(* Schneider Machine Expert - Basic project Building, file version 2.9.0.0 *)
(* ProjectInformations: Name=BUILDING *)

HARDWARE
  Cpu 0: TM221CE40T
  EthernetConfiguration: NetworkName=M221, IpAllocationMode=FixedAddress, IpAddress=0.0.0.0, SubnetMask=0.0.0.0
  SerialLineConfiguration: Baud=Baud19200, Parity=ParityEven, DataBits=DataBits8, StopBits=StopBits1, PhysicalMedium=PhysicalMediumRs485, TransmissionMode=TransmissionModeModbusRtu, SlaveId=1, Addressing=SlaveAddressing
  MastTask: UsePeriodScanMode=false, PeriodScan=100
  FastTask: Period=255
  CpuBehavior: StartingMode=StartAsPreviousState, AutoSaveRamOnEeprom=true, WatchdogPeriod=250

SYMBOLS  (address, symbol, comment, settings)
  %M0       NWDAY_HEAT_ENABLE
  %M1       WORK_MON
  %M2       WORK_TUE
  %M3       WORK_WED
  %M4       WORK_THU
  %M5       WORK_FRI
  %M6       WORK_SAT
  %M7       WORK_SUN
  %M8       IS_WORK_DAY
  %M9       IS_COLD_MONTH
  %M10      RTC_SHIFTED_FW
  %M11      RTC_SHIFTED_BW
  %M12      BEGIN_RTC_TIME_SHIFT
  %M13      INSIDE_PCYCLE
  %M14      OUTSIDE_PCYCLE
  %M17      PLOT_FULL
  %M18      ARMING
  %M19      ARMED
  %M20      TRIGGERED
  %M25      FOPEN_MAIN_DOOR  "FORCES OPEN LOBBY DOOR"
  %M26      FS_TESTING_MODE  "DISABLES CALLING FIREMEN"
  %M27      SS_TESTING_MODE  "DISABLES CALLING SECURITY"
  %M28      AUTO_LIGHTS_L
  %M29      WDONLY_LIGHTS_L  "WORK DAYS ONLY"
  %M30      BTN_ENABLE_LIGHTS_L
  %M32      AUTO_MODE_LIGHTS_L  "1=MOVEMENT 0=KEEP_ON"
  %M33      CHANGED_LIGHTS_L
  %M34      MOVEMENT_LIGHTS_L
  %M35      AUTO_LIGHTS_B
  %M36      WDONLY_LIGHTS_B
  %M37      BTN_ENABLE_LIGHTS_B
  %M39      AUTO_MODE_LIGHTS_B
  %M40      CHANGED_LIGHTS_B
  %M41      MOVEMENT_LIGHTS_B
  %M100     RFID1_REQUEST
  %M101     RFID1_RESPONSE
  %M102     RFID1_ACCEPT
  %M103     RFID1_DENIED
  %M106     RFID2_REQUEST
  %M107     RFID2_RESPONSE
  %M108     RFID2_ACCEPT
  %M109     RFID2_DENIED
  %M112     RFID3_REQUEST
  %M113     RFID3_RESPONSE
  %M114     RFID3_ACCEPT
  %M115     RFID3_DENIED
  %M118     RFID4_REQUEST
  %M119     RFID4_RESPONSE
  %M120     RFID4_ACCEPT
  %M121     RFID4_DENIED
  %M124     RFID5_REQUEST
  %M125     RFID5_RESPONSE
  %M126     PGATE_ACCEPT  "RFID5_ACCEPT"
  %M127     RFID5_DENIED
  %M128     PGATE_FOPEN  "FORCE OPEN"
  %M129     PGATE_FCLOSE  "FORCE CLOSE"
  %M199     SIM_IO  "DISABLES REAL IO"
  %M200     I00  "O3_HEATER_ENABLE"
  %M201     I01  "O3_COOLER_ENABLE"
  %M202     I02  "L_DOOR_OPENED"
  %M203     I03  "O1_DOOR_OPENED"
  %M204     I04  "O2_DOOR_OPENED"
  %M205     I05  "O3_DOOR_OPENED"
  %M206     I06  "P_GATE_OPENED"
  %M207     I07  "P_GATE_CLOSED"
  %M208     I08  "P_GATE_OBJECT"
  %M209     I09  "P_GATE_BTN"
  %M210     I10  "L_MAN_LIGHT"
  %M211     I11  "B_MAN_LIGHT"
  %M212     I12  "L_MOTION"
  %M213     I13  "C_MOTION"
  %M214     I14  "O_MOTION"
  %M215     I15  "SECURITY_KEY"
  %M216     I16  "F_ALARM_BTN"
  %M217     I17  "F_ALARM_STOP"
  %M218     I18  "O1_SMOKE"
  %M219     I19  "O2_SMOKE"
  %M220     I20  "O3_SMOKE"
  %M221     I21  "L_SMOKE"
  %M222     I22  "C1_SMOKE"
  %M223     I23  "C2_SMOKE"
  %M224     Q00  "FIRE_SIREN"
  %M225     PWM1_IN  "SCRTY_BUZZER"
  %M226     Q02  "RFID1_UNLOCK"
  %M227     Q03  "RFID2_UNLOCK"
  %M228     Q04  "RFID3_UNLOCK"
  %M229     Q05  "RFID4_UNLOCK"
  %M230     Q06  "PGATE_OPEN"
  %M231     Q07  "PGATE_CLOSE"
  %M232     Q08  "HEATER"
  %M233     Q09  "COOLER"
  %M234     Q10  "LIGHTS_L"
  %M235     Q11  "LIGHTS_B"
  %M236     Q12  "SPRINKLERS"
  %M237     Q13  "DIAL_SECURITY"
  %M238     Q14  "DIAL_FIREMEN"
  %M239     Q15  "PGATE_BULB"
  %M495     WARNING_CONFIG_ALTERED
  %M496     WARNING_AUTOSEC_IMPOSSIBLE
  %M497     WARNING_FIRE_DETECTED
  %M498     WARNING_PGATE_OPENED  "OUTSIDE PARKING CYCLE"
  %M499     WARNING_PSPOT_MISCOUNT
  %M505     ERROR_LIGHT_CONFIG
  %M506     ERROR_PGATE_FCLOPEN
  %M507     ERROR_PARKING_SPOT_CONFIG
  %M508     ERROR_TEMP_CONFIG
  %M509     ERROR_WORK_DAY_CONFIG
  %M510     ERROR_COLD_MONTH_CONFIG
  %M511     EMERGENCY
  %S50      SB_RTCUPDATE  "Set to 1, this bit allows to update the date and time"
  %SW51     SW_RTCHHMM  "RTC Function: contains in BCD HHMM: hour and minute"
  %MW0      DESIRED_TEMP
  %MW1      TOLERANCE_TEMP
  %MW2      NWDAY_DESIRED_TEMP
  %MW3      WORK_DAY_START
  %MW4      WORK_DAY_END
  %MW5      COLD_MONTH_START
  %MW6      COLD_MONTH_END
  %MW7      RTC_DESIRED_HOUR
  %MW8      PARKING_SPOT_COUNT
  %MW9      PARKING_SPOTS_TAKEN
  %MW10     PARKING_SPOT_THCOUNT  "THEORETICAL COUNT ~= <P_LOT_AREA>/11,5 (m^2)"
  %MW11     PGATE_PASSED_OBJECTS
  %MW12     PGATE_UNAUTH_OBJECTS
  %MW13     ACTIVE_SMOKE_COUNT
  %MW14     TRESHOLD_LIGHTS
  %MW15     TOLERANCE_LIGHTS
  %MW100    RFID1_REQ_START
  %MW101    RFID1_REQ_MID
  %MW102    RFID1_REQ_END
  %MW103    RFID1_RESP_START
  %MW104    RFID1_RESP_MID
  %MW105    RFID1_RESP_END
  %MW106    RFID2_REQ_START
  %MW107    RFID2_REQ_MID
  %MW108    RFID2_REQ_END
  %MW109    RFID2_RESP_START
  %MW110    RFID2_RESP_MID
  %MW111    RFID2_RESP_END
  %MW112    RFID3_REQ_START
  %MW113    RFID3_REQ_MID
  %MW114    RFID3_REQ_END
  %MW115    RFID3_RESP_START
  %MW116    RFID3_RESP_MID
  %MW117    RFID3_RESP_END
  %MW118    RFID4_REQ_START
  %MW119    RFID4_REQ_MID
  %MW120    RFID4_REQ_END
  %MW121    RFID4_RESP_START
  %MW122    RFID4_RESP_MID
  %MW123    RFID4_RESP_END
  %MW124    RFID5_REQ_START
  %MW125    RFID5_REQ_MID
  %MW126    RFID5_REQ_END
  %MW127    RFID5_RESP_START
  %MW128    RFID5_RESP_MID
  %MW129    RFID5_RESP_END
  %MW200    IW0  "MEASURED_TEMP"
  %MW201    IW1  "MEASURED_LIGHT"
  %TM0      RFID1_TM  [Type=TP, Preset=30, Base=OneHundredMilliSeconds]
  %TM1      RFID2_TM  [Type=TP, Preset=30, Base=OneHundredMilliSeconds]
  %TM2      RFID3_TM  [Type=TP, Preset=30, Base=OneHundredMilliSeconds]
  %TM3      RFID4_TM  [Type=TP, Preset=30, Base=OneHundredMilliSeconds]
  %TM4      PGATE_TM  [Preset=200, Base=OneHundredMilliSeconds]
  %TM5      ARM_TM  "60s"  [Preset=600, Base=OneHundredMilliSeconds]
  %TM6      TRIG_TM  "45s"  [Preset=450, Base=OneHundredMilliSeconds]
  %TM8      LIGHT_TM_L  [Type=TP, Preset=600, Base=OneHundredMilliSeconds]
  %TM9      LIGHT_TM_B  [Type=TP, Preset=600, Base=OneHundredMilliSeconds]
  %RTC0     RTC  [Day(Value(int=25)), Month(Value(int=3)), Year(Value(int=2000)), Hours(Value(int=0)), Minutes(Value(int=0)), Seconds(Value(int=0))]
  %I0.0     O3_HEATER_ENABLE  "OFFICE3 FL2"
  %I0.1     O3_COOLER_ENABLE  "OFFICE3 FL2"
  %I0.2     L_DOOR_OPENED  "LOBBY FL0"
  %I0.3     O1_DOOR_OPENED  "OFFICE1 FL1"
  %I0.4     O2_DOOR_OPENED  "OFFICE2 FL1"
  %I0.5     O3_DOOR_OPENED  "OFFICE3 FL3"
  %I0.6     P_GATE_OPENED  "FULLY OPENED"
  %I0.7     P_GATE_CLOSED  "FULLY CLOSED"
  %I0.8     P_GATE_OBJECT  "DETECTED OBJECT"
  %I0.9     P_GATE_BTN  "INSIDE PARKING LOT"
  %I0.10    L_MAN_LIGHT  "LOBBY"
  %I0.11    B_MAN_LIGHT  "B = C1 + C2"
  %I0.12    L_MOTION  "LOBBY SECURITY LIGHTS"
  %I0.13    C_MOTION  "CORRIDORS SECURITY LIGHTS"
  %I0.14    O_MOTION  "OFFICES SECURITY ONLY"
  %I0.15    SECURITY_KEY  "LOBBY FL0"
  %I0.16    F_ALARM_BTN  "FL0 FL1 FL2"
  %I0.17    F_ALARM_STOP  "FL0 FL1 FL2"
  %I0.18    O1_SMOKE  "OFFICE1 F1"
  %I0.19    O2_SMOKE  "OFFICE2 FL1"
  %I0.20    O3_SMOKE  "OFFICE3 FL2"
  %I0.21    L_SMOKE  "LOBBY FL0"
  %I0.22    C1_SMOKE  "CORRIDOR1 FL1"
  %I0.23    C2_SMOKE  "CORRIDOR2 FL2"
  %Q0.0     FIRE_SIREN
  %Q0.1     SCRTY_BUZZER
  %Q0.2     RFID1_UNLOCK  "LOBBY FL0"
  %Q0.3     RFID2_UNLOCK  "O1 FL1"
  %Q0.4     RFID3_UNLOCK  "O2 FL2"
  %Q0.5     RFID4_UNLOCK  "O3 FL3"
  %Q0.6     PGATE_OPEN  "PARKING LOT"
  %Q0.7     PGATE_CLOSE  "PARKING LOT"
  %Q0.8     HEATER  "O3 FL2"
  %Q0.9     COOLER  "O3 FL2"
  %Q0.10    LIGHTS_L  "LOBBY FL0"
  %Q0.11    LIGHTS_B  "B = C1 + C2"
  %Q0.12    SPRINKLERS
  %Q0.13    DIAL_SECURITY
  %Q0.14    DIAL_FIREMEN
  %Q0.15    PGATE_BULB  "IN FRONT OF PARKING LOT GATE"
  %IW0.0    MEASURED_TEMP  "-50C to +50C"  [Type=Type_0_10V, Scope=Scope_Normal, Minimum=0, Maximum=1000]
  %IW0.1    MEASURED_LIGHT  [Type=Type_0_10V, Scope=Scope_Normal, Minimum=0, Maximum=1000]
  %PWM1     BUZZER  "2kHz"  [PtoObject(RefInput=NotUsed, ZPhaseInput=NotUsed, ProbeInput=NotUsed), GlobalIndex=1, Type=PWM, TimeBase=ZeroPointOneMilliSeconds, Preset=5]

POU MAIN
  (* SectionNumber=1 *)

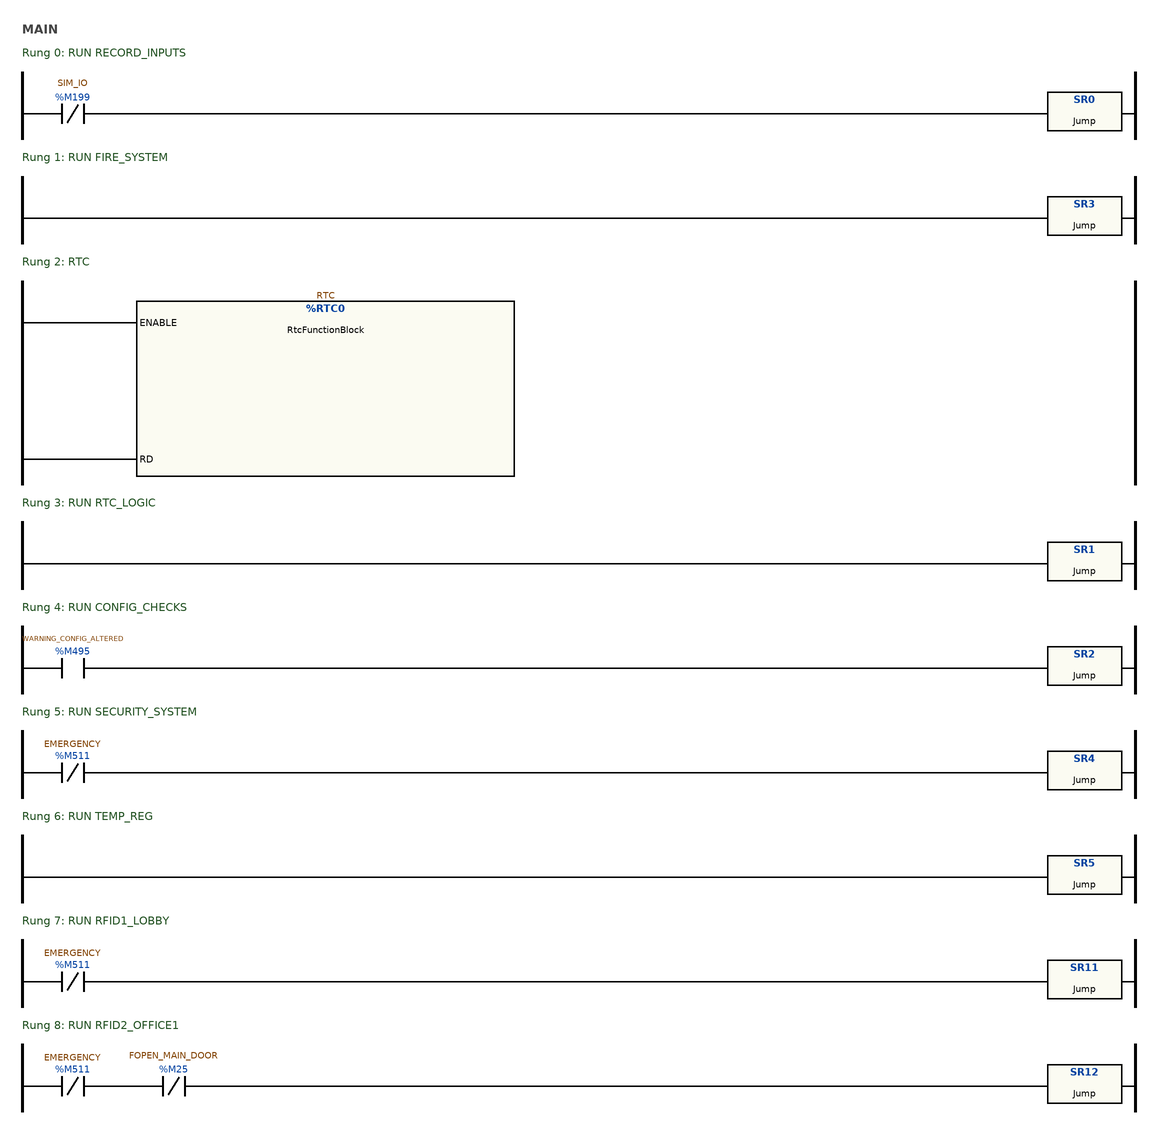

// Rung 0: RUN RECORD_INPUTS
  LDN %M199               (* SIM_IO *)
  SR0
  // as ST:
  //   IF NOT SIM_IO THEN SR0(); END_IF;

// Rung 1: RUN FIRE_SYSTEM
  LD 1
  SR3
  // as ST:
  //   SR3();

// Rung 2: RTC
  BLK %RTC0               (* RTC *)
  LD 1
  ENABLE
  LD 1
  RD
  END_BLK
  // as ST:
  //   RTC(ENABLE := TRUE, RD := TRUE);

// Rung 3: RUN RTC_LOGIC
  LD 1
  SR1
  // as ST:
  //   SR1();

// Rung 4: RUN CONFIG_CHECKS
  LD %M495                (* WARNING_CONFIG_ALTERED *)
  SR2
  // as ST:
  //   IF WARNING_CONFIG_ALTERED THEN SR2(); END_IF;

// Rung 5: RUN SECURITY_SYSTEM
  LDN %M511               (* EMERGENCY *)
  SR4
  // as ST:
  //   IF NOT EMERGENCY THEN SR4(); END_IF;

// Rung 6: RUN TEMP_REG
  LD 1
  SR5
  // as ST:
  //   SR5();

// Rung 7: RUN RFID1_LOBBY
  LDN %M511               (* EMERGENCY *)
  SR11
  // as ST:
  //   IF NOT EMERGENCY THEN SR11(); END_IF;

// Rung 8: RUN RFID2_OFFICE1
  LDN %M511               (* EMERGENCY *)
  ANDN %M25               (* FOPEN_MAIN_DOOR *)
  SR12
  // as ST:
  //   IF NOT EMERGENCY AND NOT FOPEN_MAIN_DOOR THEN SR12(); END_IF;

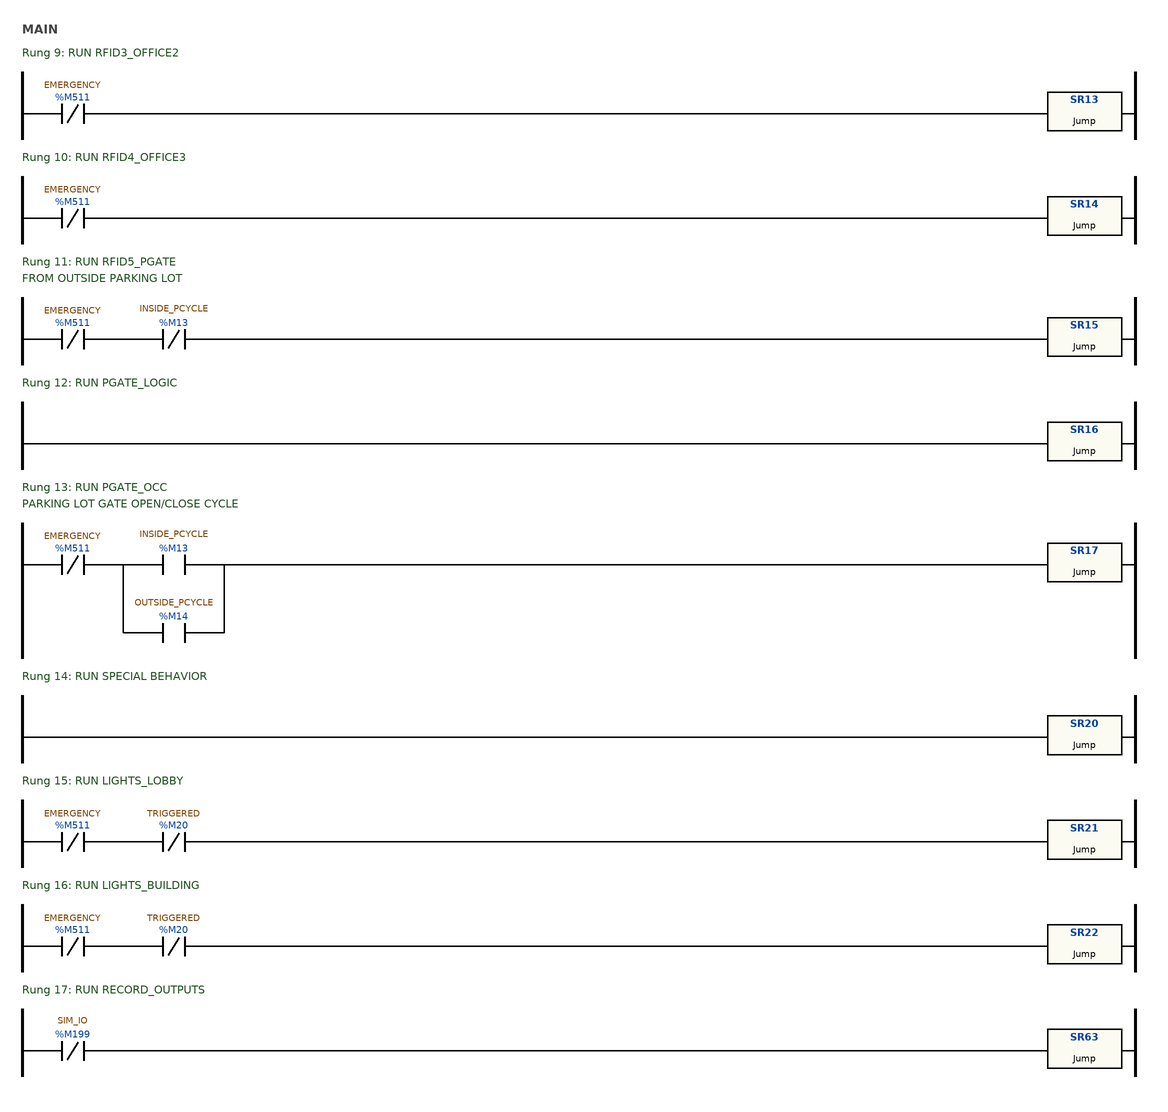

// Rung 9: RUN RFID3_OFFICE2
  LDN %M511               (* EMERGENCY *)
  SR13
  // as ST:
  //   IF NOT EMERGENCY THEN SR13(); END_IF;

// Rung 10: RUN RFID4_OFFICE3
  LDN %M511               (* EMERGENCY *)
  SR14
  // as ST:
  //   IF NOT EMERGENCY THEN SR14(); END_IF;

// Rung 11: RUN RFID5_PGATE
// FROM OUTSIDE PARKING LOT
  LDN %M511               (* EMERGENCY *)
  ANDN %M13               (* INSIDE_PCYCLE *)
  SR15
  // as ST:
  //   IF NOT EMERGENCY AND NOT INSIDE_PCYCLE THEN SR15(); END_IF;

// Rung 12: RUN PGATE_LOGIC
  LD 1
  SR16
  // as ST:
  //   SR16();

// Rung 13: RUN PGATE_OCC
// PARKING LOT GATE OPEN/CLOSE CYCLE
  LDN %M511               (* EMERGENCY *)
  AND( %M13               (* INSIDE_PCYCLE *)
  OR %M14                 (* OUTSIDE_PCYCLE *)
  )
  SR17
  // as ST:
  //   IF NOT EMERGENCY AND (INSIDE_PCYCLE OR OUTSIDE_PCYCLE) THEN SR17(); END_IF;

// Rung 14: RUN SPECIAL BEHAVIOR
  LD 1
  SR20
  // as ST:
  //   SR20();

// Rung 15: RUN LIGHTS_LOBBY
  LDN %M511               (* EMERGENCY *)
  ANDN %M20               (* TRIGGERED *)
  SR21
  // as ST:
  //   IF NOT EMERGENCY AND NOT TRIGGERED THEN SR21(); END_IF;

// Rung 16: RUN LIGHTS_BUILDING
  LDN %M511               (* EMERGENCY *)
  ANDN %M20               (* TRIGGERED *)
  SR22
  // as ST:
  //   IF NOT EMERGENCY AND NOT TRIGGERED THEN SR22(); END_IF;

// Rung 17: RUN RECORD_OUTPUTS
  LDN %M199               (* SIM_IO *)
  SR63
  // as ST:
  //   IF NOT SIM_IO THEN SR63(); END_IF;

Subroutine RECORD_INPUTS
  (* SectionNumber=2, Number=0 *)

// Rung 18: %I0.0 TO I00
  LD %I0.0                (* O3_HEATER_ENABLE *)
  ST %M200                (* I00 *)
  // as ST:
  //   I00 := O3_HEATER_ENABLE;

// Rung 19: %I0.1 TO I01
  LD %I0.1                (* O3_COOLER_ENABLE *)
  ST %M201                (* I01 *)
  // as ST:
  //   I01 := O3_COOLER_ENABLE;

// Rung 20: %I0.2 TO I02
  LD %I0.2                (* L_DOOR_OPENED *)
  ST %M202                (* I02 *)
  // as ST:
  //   I02 := L_DOOR_OPENED;

// Rung 21: %I0.3 TO I03
  LD %I0.3                (* O1_DOOR_OPENED *)
  ST %M203                (* I03 *)
  // as ST:
  //   I03 := O1_DOOR_OPENED;

// Rung 22: %I0.4 TO I04
  LD %I0.4                (* O2_DOOR_OPENED *)
  ST %M204                (* I04 *)
  // as ST:
  //   I04 := O2_DOOR_OPENED;

// Rung 23: %I0.5 TO I05
  LD %I0.5                (* O3_DOOR_OPENED *)
  ST %M205                (* I05 *)
  // as ST:
  //   I05 := O3_DOOR_OPENED;

// Rung 24: %I0.6 TO I06
  LD %I0.6                (* P_GATE_OPENED *)
  ST %M206                (* I06 *)
  // as ST:
  //   I06 := P_GATE_OPENED;

// Rung 25: %I0.7 TO I07
  LD %I0.7                (* P_GATE_CLOSED *)
  ST %M207                (* I07 *)
  // as ST:
  //   I07 := P_GATE_CLOSED;

// Rung 26: %I0.8 TO I08
  LD %I0.8                (* P_GATE_OBJECT *)
  ST %M208                (* I08 *)
  // as ST:
  //   I08 := P_GATE_OBJECT;

// Rung 27: %I0.9 TO I09
  LD %I0.9                (* P_GATE_BTN *)
  ST %M209                (* I09 *)
  // as ST:
  //   I09 := P_GATE_BTN;

// Rung 28: %I0.10 TO I10
  LD %I0.10               (* L_MAN_LIGHT *)
  ST %M210                (* I10 *)
  // as ST:
  //   I10 := L_MAN_LIGHT;

// Rung 29: %I0.11 TO I11
  LD %I0.11               (* B_MAN_LIGHT *)
  ST %M211                (* I11 *)
  // as ST:
  //   I11 := B_MAN_LIGHT;

// Rung 30: %I0.12 TO I12
  LD %I0.12               (* L_MOTION *)
  ST %M212                (* I12 *)
  // as ST:
  //   I12 := L_MOTION;

// Rung 31: %I0.13 TO I13
  LD %I0.13               (* C_MOTION *)
  ST %M213                (* I13 *)
  // as ST:
  //   I13 := C_MOTION;

// Rung 32: %I0.14 TO I14
  LD %I0.14               (* O_MOTION *)
  ST %M214                (* I14 *)
  // as ST:
  //   I14 := O_MOTION;

// Rung 33: %I0.15 TO I15
  LD %I0.15               (* SECURITY_KEY *)
  ST %M215                (* I15 *)
  // as ST:
  //   I15 := SECURITY_KEY;

// Rung 34: %I0.16 TO I16
  LD %I0.16               (* F_ALARM_BTN *)
  ST %M216                (* I16 *)
  // as ST:
  //   I16 := F_ALARM_BTN;

// Rung 35: %I0.17 TO I17
  LD %I0.17               (* F_ALARM_STOP *)
  ST %M217                (* I17 *)
  // as ST:
  //   I17 := F_ALARM_STOP;

// Rung 36: %I0.18 TO I18
  LD %I0.18               (* O1_SMOKE *)
  ST %M218                (* I18 *)
  // as ST:
  //   I18 := O1_SMOKE;

// Rung 37: %I0.19 TO I19
  LD %I0.19               (* O2_SMOKE *)
  ST %M219                (* I19 *)
  // as ST:
  //   I19 := O2_SMOKE;

// Rung 38: %I0.20 TO I20
  LD %I0.20               (* O3_SMOKE *)
  ST %M220                (* I20 *)
  // as ST:
  //   I20 := O3_SMOKE;

// Rung 39: %I0.21 TO I21
  LD %I0.21               (* L_SMOKE *)
  ST %M221                (* I21 *)
  // as ST:
  //   I21 := L_SMOKE;

// Rung 40: %I0.22 TO I22
  LD %I0.22               (* C1_SMOKE *)
  ST %M222                (* I22 *)
  // as ST:
  //   I22 := C1_SMOKE;

// Rung 41: %I0.23 TO I23
  LD %I0.23               (* C2_SMOKE *)
  ST %M223                (* I23 *)
  // as ST:
  //   I23 := C2_SMOKE;

// Rung 42: %IW0.0 TO IW0
  LD 1
  [ %MW200 := %IW0.0 ]    (* IW0, MEASURED_TEMP *)
  // as ST:
  //   IW0 := MEASURED_TEMP;

// Rung 43: %IW0.1 TO IW1
  LD 1
  [ %MW201 := %IW0.1 ]    (* IW1, MEASURED_LIGHT *)
  // as ST:
  //   IW1 := MEASURED_LIGHT;

Subroutine RTC_LOGIC
  (* SectionNumber=3, Number=1 *)

// Rung 44: RTC DST FORWARD SHIFT REQUEST
  LDN %M10                (* RTC_SHIFTED_FW *)
  AND [ %RTC0.HOURS = 3 ] (* RTC *)
  AND [ %RTC0.MINUTES = 0 ](* RTC *)
  AND [ %RTC0.SECONDS = 0 ](* RTC *)
  AND [ %RTC0.MONTH = 3 ] (* RTC *)
  AND [ %RTC0.DAY >= 25 ] (* RTC *)
  AND [ %RTC0.DAYOFWEEK = 7 ](* RTC *)
  S %M10                  (* RTC_SHIFTED_FW *)
  R %M11                  (* RTC_SHIFTED_BW *)
  [ %MW7 := 1024 ]        (* RTC_DESIRED_HOUR *)
  // as ST:
  //   _t1 := NOT RTC_SHIFTED_FW AND RTC.HOURS = 3 AND RTC.MINUTES = 0 AND RTC.SECONDS = 0 AND RTC.MONTH = 3 AND RTC.DAY >= 25 AND RTC.DAYOFWEEK = 7;
  //   IF _t1 THEN RTC_SHIFTED_FW := TRUE; END_IF;
  //   IF _t1 THEN RTC_SHIFTED_BW := FALSE; END_IF;
  //   IF _t1 THEN RTC_DESIRED_HOUR := 1024; END_IF;

// Rung 45: RTC DST BACKWARD SHIFT REQUEST
  LDN %M11                (* RTC_SHIFTED_BW *)
  AND [ %RTC0.HOURS = 4 ] (* RTC *)
  AND [ %RTC0.MINUTES = 0 ](* RTC *)
  AND [ %RTC0.SECONDS = 0 ](* RTC *)
  AND [ %RTC0.MONTH = 10 ](* RTC *)
  AND [ %RTC0.DAY >= 25 ] (* RTC *)
  AND [ %RTC0.DAYOFWEEK = 7 ](* RTC *)
  S %M11                  (* RTC_SHIFTED_BW *)
  R %M10                  (* RTC_SHIFTED_FW *)
  [ %MW7 := 768 ]         (* RTC_DESIRED_HOUR *)
  // as ST:
  //   _t1 := NOT RTC_SHIFTED_BW AND RTC.HOURS = 4 AND RTC.MINUTES = 0 AND RTC.SECONDS = 0 AND RTC.MONTH = 10 AND RTC.DAY >= 25 AND RTC.DAYOFWEEK = 7;
  //   IF _t1 THEN RTC_SHIFTED_BW := TRUE; END_IF;
  //   IF _t1 THEN RTC_SHIFTED_FW := FALSE; END_IF;
  //   IF _t1 THEN RTC_DESIRED_HOUR := 768; END_IF;

// Rung 46: RTC TIME SHIFT EXECUTE
  LDR %M10                (* RTC_SHIFTED_FW *)
  ORR %M11                (* RTC_SHIFTED_BW *)
  ST %S50                 (* SB_RTCUPDATE *)
  [ %SW51 := %MW7 ]       (* SW_RTCHHMM, RTC_DESIRED_HOUR *)
  // as ST:
  //   SB_RTCUPDATE := RISING(RTC_SHIFTED_FW) OR RISING(RTC_SHIFTED_BW);
  //   IF RISING(RTC_SHIFTED_FW) OR RISING(RTC_SHIFTED_BW) THEN SW_RTCHHMM := RTC_DESIRED_HOUR; END_IF;

// Rung 47: WORK DAY CHECK
  LDN %M509               (* ERROR_WORK_DAY_CONFIG *)
  AND( %M1                (* WORK_MON *)
  AND [ %RTC0.DAYOFWEEK = 1 ](* RTC *)
  OR( %M2                 (* WORK_TUE *)
  AND [ %RTC0.DAYOFWEEK = 2 ](* RTC *)
  )
  OR( %M3                 (* WORK_WED *)
  AND [ %RTC0.DAYOFWEEK = 3 ](* RTC *)
  )
  OR( %M4                 (* WORK_THU *)
  AND [ %RTC0.DAYOFWEEK = 4 ](* RTC *)
  )
  OR( %M5                 (* WORK_FRI *)
  AND [ %RTC0.DAYOFWEEK = 5 ](* RTC *)
  )
  OR( %M6                 (* WORK_SAT *)
  AND [ %RTC0.DAYOFWEEK = 6 ](* RTC *)
  )
  OR( %M7                 (* WORK_SUN *)
  AND [ %RTC0.DAYOFWEEK = 7 ](* RTC *)
  )
  )
  AND [ %RTC0.HOURS >= %MW3 ](* RTC, WORK_DAY_START *)
  AND [ %RTC0.HOURS <= %MW4 ](* RTC, WORK_DAY_END *)
  ST %M8                  (* IS_WORK_DAY *)
  // as ST:
  //   IS_WORK_DAY := NOT ERROR_WORK_DAY_CONFIG AND (WORK_MON AND RTC.DAYOFWEEK = 1 OR WORK_TUE AND RTC.DAYOFWEEK = 2 OR WORK_WED AND RTC.DAYOFWEEK = 3 OR WORK_THU AND RTC.DAYOFWEEK = 4 OR WORK_FRI AND RTC.DAYOFWEEK = 5 OR WORK_SAT AND RTC.DAYOFWEEK = 6 OR WORK_SUN AND RTC.DAYOFWEEK = 7) AND RTC.HOURS >= WORK_DAY_START AND RTC.HOURS <= WORK_DAY_END;

Subroutine CONFIG_CHECKS
  (* SectionNumber=4, Number=2 *)

// Rung 48: COLD MONTH CONFIG ERROR
  LD %M0                  (* NWDAY_HEAT_ENABLE *)
  MPS
  AND [ %MW5 >= 1 ]       (* COLD_MONTH_START *)
  AND [ %MW5 <= 12 ]      (* COLD_MONTH_START *)
  AND [ %MW6 >= 1 ]       (* COLD_MONTH_END *)
  AND [ %MW6 <= 12 ]      (* COLD_MONTH_END *)
  R %M510                 (* ERROR_COLD_MONTH_CONFIG *)
  MPP
  AND( [ %MW5 < 1 ]       (* COLD_MONTH_START *)
  OR [ %MW5 > 12 ]        (* COLD_MONTH_START *)
  OR [ %MW6 < 1 ]         (* COLD_MONTH_END *)
  OR [ %MW6 > 12 ]        (* COLD_MONTH_END *)
  )
  S %M510                 (* ERROR_COLD_MONTH_CONFIG *)
  // as ST:
  //   IF NWDAY_HEAT_ENABLE AND COLD_MONTH_START >= 1 AND COLD_MONTH_START <= 12 AND COLD_MONTH_END >= 1 AND COLD_MONTH_END <= 12 THEN ERROR_COLD_MONTH_CONFIG := FALSE; END_IF;
  //   IF NWDAY_HEAT_ENABLE AND (COLD_MONTH_START < 1 OR COLD_MONTH_START > 12 OR COLD_MONTH_END < 1 OR COLD_MONTH_END > 12) THEN ERROR_COLD_MONTH_CONFIG := TRUE; END_IF;

// Rung 49: WORK DAY CONFIG ERROR
  LD %M1                  (* WORK_MON *)
  OR %M2                  (* WORK_TUE *)
  OR %M3                  (* WORK_WED *)
  OR %M4                  (* WORK_THU *)
  OR %M5                  (* WORK_FRI *)
  OR %M6                  (* WORK_SAT *)
  OR %M7                  (* WORK_SUN *)
  MPS
  AND [ %MW3 > 0 ]        (* WORK_DAY_START *)
  AND [ %MW4 > 0 ]        (* WORK_DAY_END *)
  AND [ %MW3 < 24 ]       (* WORK_DAY_START *)
  AND [ %MW4 < 24 ]       (* WORK_DAY_END *)
  AND [ %MW3 <= %MW4 ]    (* WORK_DAY_START, WORK_DAY_END *)
  R %M509                 (* ERROR_WORK_DAY_CONFIG *)
  MPP
  AND( [ %MW3 < 0 ]       (* WORK_DAY_START *)
  OR [ %MW4 < 0 ]         (* WORK_DAY_END *)
  OR [ %MW3 >= 24 ]       (* WORK_DAY_START *)
  OR [ %MW4 >= 24 ]       (* WORK_DAY_END *)
  OR [ %MW3 > %MW4 ]      (* WORK_DAY_START, WORK_DAY_END *)
  )
  S %M509                 (* ERROR_WORK_DAY_CONFIG *)
  // as ST:
  //   IF (WORK_MON OR WORK_TUE OR WORK_WED OR WORK_THU OR WORK_FRI OR WORK_SAT OR WORK_SUN) AND WORK_DAY_START > 0 AND WORK_DAY_END > 0 AND WORK_DAY_START < 24 AND WORK_DAY_END < 24 AND WORK_DAY_START <= WORK_DAY_END THEN ERROR_WORK_DAY_CONFIG := FALSE; END_IF;
  //   IF (WORK_MON OR WORK_TUE OR WORK_WED OR WORK_THU OR WORK_FRI OR WORK_SAT OR WORK_SUN) AND (WORK_DAY_START < 0 OR WORK_DAY_END < 0 OR WORK_DAY_START >= 24 OR WORK_DAY_END >= 24 OR WORK_DAY_START > WORK_DAY_END) THEN ERROR_WORK_DAY_CONFIG := TRUE; END_IF;

// Rung 50: WORK DAY NOT CONFIGURED
  LDN %M1                 (* WORK_MON *)
  ANDN %M2                (* WORK_TUE *)
  ANDN %M3                (* WORK_WED *)
  ANDN %M4                (* WORK_THU *)
  ANDN %M5                (* WORK_FRI *)
  ANDN %M6                (* WORK_SAT *)
  ANDN %M7                (* WORK_SUN *)
  R %M509                 (* ERROR_WORK_DAY_CONFIG *)
  // as ST:
  //   IF NOT WORK_MON AND NOT WORK_TUE AND NOT WORK_WED AND NOT WORK_THU AND NOT WORK_FRI AND NOT WORK_SAT AND NOT WORK_SUN THEN ERROR_WORK_DAY_CONFIG := FALSE; END_IF;

// Rung 51: WORK DAY TEMP CONFIG ERROR
  LD %M1                  (* WORK_MON *)
  OR %M2                  (* WORK_TUE *)
  OR %M3                  (* WORK_WED *)
  OR %M4                  (* WORK_THU *)
  OR %M5                  (* WORK_FRI *)
  OR %M6                  (* WORK_SAT *)
  OR %M7                  (* WORK_SUN *)
  MPS
  AND [ %MW0 >= 0 ]       (* DESIRED_TEMP *)
  AND [ %MW0 <= 1000 ]    (* DESIRED_TEMP *)
  AND [ %MW0 + %MW1 <= 1000 ](* DESIRED_TEMP, TOLERANCE_TEMP *)
  AND [ %MW0 - %MW1 >= 0 ](* DESIRED_TEMP, TOLERANCE_TEMP *)
  R %M508                 (* ERROR_TEMP_CONFIG *)
  MPP
  AND( [ %MW0 < 0 ]       (* DESIRED_TEMP *)
  OR [ %MW0 > 1000 ]      (* DESIRED_TEMP *)
  OR [ %MW0 + %MW1 > 1000 ](* DESIRED_TEMP, TOLERANCE_TEMP *)
  OR [ %MW0 - %MW1 < 0 ]  (* DESIRED_TEMP, TOLERANCE_TEMP *)
  )
  S %M508                 (* ERROR_TEMP_CONFIG *)
  // as ST:
  //   IF (WORK_MON OR WORK_TUE OR WORK_WED OR WORK_THU OR WORK_FRI OR WORK_SAT OR WORK_SUN) AND DESIRED_TEMP >= 0 AND DESIRED_TEMP <= 1000 AND DESIRED_TEMP + TOLERANCE_TEMP <= 1000 AND DESIRED_TEMP - TOLERANCE_TEMP >= 0 THEN ERROR_TEMP_CONFIG := FALSE; END_IF;
  //   IF (WORK_MON OR WORK_TUE OR WORK_WED OR WORK_THU OR WORK_FRI OR WORK_SAT OR WORK_SUN) AND (DESIRED_TEMP < 0 OR DESIRED_TEMP > 1000 OR DESIRED_TEMP + TOLERANCE_TEMP > 1000 OR DESIRED_TEMP - TOLERANCE_TEMP < 0) THEN ERROR_TEMP_CONFIG := TRUE; END_IF;

// Rung 52: NON WORK DAY TEMP CONFIG ERROR
  LD %M0                  (* NWDAY_HEAT_ENABLE *)
  MPS
  AND [ %MW2 >= 0 ]       (* NWDAY_DESIRED_TEMP *)
  AND [ %MW2 <= 1000 ]    (* NWDAY_DESIRED_TEMP *)
  AND [ %MW2 + %MW1 <= 1000 ](* NWDAY_DESIRED_TEMP, TOLERANCE_TEMP *)
  AND [ %MW2 - %MW1 >= 0 ](* NWDAY_DESIRED_TEMP, TOLERANCE_TEMP *)
  R %M508                 (* ERROR_TEMP_CONFIG *)
  MPP
  AND( [ %MW2 < 0 ]       (* NWDAY_DESIRED_TEMP *)
  OR [ %MW2 > 1000 ]      (* NWDAY_DESIRED_TEMP *)
  OR [ %MW2 + %MW1 > 1000 ](* NWDAY_DESIRED_TEMP, TOLERANCE_TEMP *)
  OR [ %MW2 - %MW1 < 0 ]  (* NWDAY_DESIRED_TEMP, TOLERANCE_TEMP *)
  )
  S %M508                 (* ERROR_TEMP_CONFIG *)
  // as ST:
  //   IF NWDAY_HEAT_ENABLE AND NWDAY_DESIRED_TEMP >= 0 AND NWDAY_DESIRED_TEMP <= 1000 AND NWDAY_DESIRED_TEMP + TOLERANCE_TEMP <= 1000 AND NWDAY_DESIRED_TEMP - TOLERANCE_TEMP >= 0 THEN ERROR_TEMP_CONFIG := FALSE; END_IF;
  //   IF NWDAY_HEAT_ENABLE AND (NWDAY_DESIRED_TEMP < 0 OR NWDAY_DESIRED_TEMP > 1000 OR NWDAY_DESIRED_TEMP + TOLERANCE_TEMP > 1000 OR NWDAY_DESIRED_TEMP - TOLERANCE_TEMP < 0) THEN ERROR_TEMP_CONFIG := TRUE; END_IF;

// Rung 53: DESIRED LIGHT CONFIG ERROR
  LD %M28                 (* AUTO_LIGHTS_L *)
  OR %M35                 (* AUTO_LIGHTS_B *)
  MPS
  AND [ %MW14 >= 0 ]      (* TRESHOLD_LIGHTS *)
  AND [ %MW14 <= 1000 ]   (* TRESHOLD_LIGHTS *)
  AND [ %MW14 - %MW15 >= 0 ](* TRESHOLD_LIGHTS, TOLERANCE_LIGHTS *)
  AND [ %MW14 + %MW15 <= 1000 ](* TRESHOLD_LIGHTS, TOLERANCE_LIGHTS *)
  R %M505                 (* ERROR_LIGHT_CONFIG *)
  MPP
  AND( [ %MW14 < 0 ]      (* TRESHOLD_LIGHTS *)
  OR [ %MW14 > 1000 ]     (* TRESHOLD_LIGHTS *)
  OR [ %MW14 - %MW15 < 0 ](* TRESHOLD_LIGHTS, TOLERANCE_LIGHTS *)
  OR [ %MW14 + %MW15 > 1000 ](* TRESHOLD_LIGHTS, TOLERANCE_LIGHTS *)
  )
  S %M505                 (* ERROR_LIGHT_CONFIG *)
  // as ST:
  //   IF (AUTO_LIGHTS_L OR AUTO_LIGHTS_B) AND TRESHOLD_LIGHTS >= 0 AND TRESHOLD_LIGHTS <= 1000 AND TRESHOLD_LIGHTS - TOLERANCE_LIGHTS >= 0 AND TRESHOLD_LIGHTS + TOLERANCE_LIGHTS <= 1000 THEN ERROR_LIGHT_CONFIG := FALSE; END_IF;
  //   IF (AUTO_LIGHTS_L OR AUTO_LIGHTS_B) AND (TRESHOLD_LIGHTS < 0 OR TRESHOLD_LIGHTS > 1000 OR TRESHOLD_LIGHTS - TOLERANCE_LIGHTS < 0 OR TRESHOLD_LIGHTS + TOLERANCE_LIGHTS > 1000) THEN ERROR_LIGHT_CONFIG := TRUE; END_IF;

// Rung 54: PARKING SPOT CONFIG ERROR
  LD [ %MW8 > %MW10 ]     (* PARKING_SPOT_COUNT, PARKING_SPOT_THCOUNT *)
  OR [ %MW8 < 0 ]         (* PARKING_SPOT_COUNT *)
  OR [ %MW10 < 0 ]        (* PARKING_SPOT_THCOUNT *)
  OR [ %MW9 < 0 ]         (* PARKING_SPOTS_TAKEN *)
  OR [ %MW9 > %MW10 ]     (* PARKING_SPOTS_TAKEN, PARKING_SPOT_THCOUNT *)
  S %M507                 (* ERROR_PARKING_SPOT_CONFIG *)
  // as ST:
  //   IF PARKING_SPOT_COUNT > PARKING_SPOT_THCOUNT OR PARKING_SPOT_COUNT < 0 OR PARKING_SPOT_THCOUNT < 0 OR PARKING_SPOTS_TAKEN < 0 OR PARKING_SPOTS_TAKEN > PARKING_SPOT_THCOUNT THEN ERROR_PARKING_SPOT_CONFIG := TRUE; END_IF;

// Rung 55: PARKING SPOT CONFIG NO ERROR
  LD [ %MW8 <= %MW10 ]    (* PARKING_SPOT_COUNT, PARKING_SPOT_THCOUNT *)
  AND [ %MW8 >= 0 ]       (* PARKING_SPOT_COUNT *)
  AND [ %MW10 >= 0 ]      (* PARKING_SPOT_THCOUNT *)
  AND [ %MW9 >= 0 ]       (* PARKING_SPOTS_TAKEN *)
  AND [ %MW8 <= %MW10 ]   (* PARKING_SPOT_COUNT, PARKING_SPOT_THCOUNT *)
  R %M507                 (* ERROR_PARKING_SPOT_CONFIG *)
  // as ST:
  //   IF PARKING_SPOT_COUNT <= PARKING_SPOT_THCOUNT AND PARKING_SPOT_COUNT >= 0 AND PARKING_SPOT_THCOUNT >= 0 AND PARKING_SPOTS_TAKEN >= 0 AND PARKING_SPOT_COUNT <= PARKING_SPOT_THCOUNT THEN ERROR_PARKING_SPOT_CONFIG := FALSE; END_IF;

// Rung 56: REMOVE PARKING SPOT MISCOUNT WARNING
  LDN %M507               (* ERROR_PARKING_SPOT_CONFIG *)
  AND %M499               (* WARNING_PSPOT_MISCOUNT *)
  R %M499                 (* WARNING_PSPOT_MISCOUNT *)
  // as ST:
  //   IF NOT ERROR_PARKING_SPOT_CONFIG AND WARNING_PSPOT_MISCOUNT THEN WARNING_PSPOT_MISCOUNT := FALSE; END_IF;

// Rung 57: CONFIG CHECKED
  LD 1
  R %M495                 (* WARNING_CONFIG_ALTERED *)
  // as ST:
  //   WARNING_CONFIG_ALTERED := FALSE;

Subroutine FIRE_SYSTEM
  (* SectionNumber=5, Number=3 *)

// Rung 58: SMOKE SIGNAL
  LDR %M223               (* I23 *)
  ORR %M222               (* I22 *)
  ORR %M218               (* I18 *)
  ORR %M219               (* I19 *)
  ORR %M221               (* I21 *)
  ORR %M220               (* I20 *)
  ORR %M216               (* I16 *)
  MPS
  S %M497                 (* WARNING_FIRE_DETECTED *)
  MPP
  ANDN %M26               (* FS_TESTING_MODE *)
  S %M238                 (* Q14 *)
  // as ST:
  //   IF RISING(I23) OR RISING(I22) OR RISING(I18) OR RISING(I19) OR RISING(I21) OR RISING(I20) OR RISING(I16) THEN WARNING_FIRE_DETECTED := TRUE; END_IF;
  //   IF (RISING(I23) OR RISING(I22) OR RISING(I18) OR RISING(I19) OR RISING(I21) OR RISING(I20) OR RISING(I16)) AND NOT FS_TESTING_MODE THEN Q14 := TRUE; END_IF;

// Rung 59: INCREMENT ACTIVE SMOKE SIGNALS
  LDR %M223               (* I23 *)
  ORR %M222               (* I22 *)
  ORR %M218               (* I18 *)
  ORR %M219               (* I19 *)
  ORR %M221               (* I21 *)
  ORR %M220               (* I20 *)
  [ %MW13 := %MW13 + 1 ]  (* ACTIVE_SMOKE_COUNT, ACTIVE_SMOKE_COUNT *)
  // as ST:
  //   IF RISING(I23) OR RISING(I22) OR RISING(I18) OR RISING(I19) OR RISING(I21) OR RISING(I20) THEN ACTIVE_SMOKE_COUNT := ACTIVE_SMOKE_COUNT + 1; END_IF;

// Rung 60: DECREMENT ACTIVE SMOKE SIGNALS
  LDF %M223               (* I23 *)
  ORF %M222               (* I22 *)
  ORF %M218               (* I18 *)
  ORF %M219               (* I19 *)
  ORF %M221               (* I21 *)
  ORF %M220               (* I20 *)
  [ %MW13 := %MW13 - 1 ]  (* ACTIVE_SMOKE_COUNT, ACTIVE_SMOKE_COUNT *)
  // as ST:
  //   IF FALLING(I23) OR FALLING(I22) OR FALLING(I18) OR FALLING(I19) OR FALLING(I21) OR FALLING(I20) THEN ACTIVE_SMOKE_COUNT := ACTIVE_SMOKE_COUNT - 1; END_IF;

// Rung 61: RAISE EMERGENCY FLAG
// SMOKE IN MULTIPLE LOCATIONS
  LD %M497                (* WARNING_FIRE_DETECTED *)
  AND [ %MW13 > 1 ]       (* ACTIVE_SMOKE_COUNT *)
  MPS
  S %M511                 (* EMERGENCY *)
  MPP
  ANDN %M26               (* FS_TESTING_MODE *)
  S %M236                 (* Q12 *)
  // as ST:
  //   IF WARNING_FIRE_DETECTED AND ACTIVE_SMOKE_COUNT > 1 THEN EMERGENCY := TRUE; END_IF;
  //   IF WARNING_FIRE_DETECTED AND ACTIVE_SMOKE_COUNT > 1 AND NOT FS_TESTING_MODE THEN Q12 := TRUE; END_IF;

// Rung 62: DISENGAGE SPRINKLERS
  LD %M497                (* WARNING_FIRE_DETECTED *)
  AND [ %MW13 = 0 ]       (* ACTIVE_SMOKE_COUNT *)
  ORF %M497               (* WARNING_FIRE_DETECTED *)
  R %M236                 (* Q12 *)
  // as ST:
  //   IF WARNING_FIRE_DETECTED AND ACTIVE_SMOKE_COUNT = 0 OR FALLING(WARNING_FIRE_DETECTED) THEN Q12 := FALSE; END_IF;

// Rung 63: LOWER EMERGENCY FLAG
  LDF %M497               (* WARNING_FIRE_DETECTED *)
  R %M511                 (* EMERGENCY *)
  // as ST:
  //   IF FALLING(WARNING_FIRE_DETECTED) THEN EMERGENCY := FALSE; END_IF;

// Rung 64: TURN ON FIRE ALARM
  LD %M497                (* WARNING_FIRE_DETECTED *)
  ST %M224                (* Q00 *)
  // as ST:
  //   Q00 := WARNING_FIRE_DETECTED;

// Rung 65: STOP ALARM WITH BUTTON
  LDR %I0.17              (* F_ALARM_STOP *)
  ANDN %I0.23             (* C2_SMOKE *)
  ANDN %I0.22             (* C1_SMOKE *)
  ANDN %I0.21             (* L_SMOKE *)
  ANDN %I0.18             (* O1_SMOKE *)
  ANDN %I0.19             (* O2_SMOKE *)
  ANDN %I0.20             (* O3_SMOKE *)
  ANDN %I0.16             (* F_ALARM_BTN *)
  R %M497                 (* WARNING_FIRE_DETECTED *)
  R %M238                 (* Q14 *)
  // as ST:
  //   IF RISING(F_ALARM_STOP) AND NOT C2_SMOKE AND NOT C1_SMOKE AND NOT L_SMOKE AND NOT O1_SMOKE AND NOT O2_SMOKE AND NOT O3_SMOKE AND NOT F_ALARM_BTN THEN WARNING_FIRE_DETECTED := FALSE; END_IF;
  //   IF RISING(F_ALARM_STOP) AND NOT C2_SMOKE AND NOT C1_SMOKE AND NOT L_SMOKE AND NOT O1_SMOKE AND NOT O2_SMOKE AND NOT O3_SMOKE AND NOT F_ALARM_BTN THEN Q14 := FALSE; END_IF;

Subroutine SECURITY_SYSTEM
  (* SectionNumber=6, Number=4 *)

// Rung 66: START ARMING SYSTEM
  LDR %I0.15              (* SECURITY_KEY *)
  S %M18                  (* ARMING *)
  // as ST:
  //   IF RISING(SECURITY_KEY) THEN ARMING := TRUE; END_IF;

// Rung 67: ARM SYSTEM
  BLK %TM5                (* ARM_TM *)
  LD %M18                 (* ARMING *)
  IN
  OUT_BLK
  LD Q
  R %M18                  (* ARMING *)
  S %M19                  (* ARMED *)
  END_BLK
  // as ST:
  //   ARM_TM(IN := ARMING);
  //   IF ARM_TM.Q THEN ARMING := FALSE; END_IF;
  //   IF ARM_TM.Q THEN ARMED := TRUE; END_IF;

// Rung 68: DISARM SYSTEM
  LDF %I0.15              (* SECURITY_KEY *)
  R %M18                  (* ARMING *)
  R %M19                  (* ARMED *)
  R %M20                  (* TRIGGERED *)
  // as ST:
  //   IF FALLING(SECURITY_KEY) THEN ARMING := FALSE; END_IF;
  //   IF FALLING(SECURITY_KEY) THEN ARMED := FALSE; END_IF;
  //   IF FALLING(SECURITY_KEY) THEN TRIGGERED := FALSE; END_IF;

// Rung 69: READ DETECTION SIGNALS
  LD %M202                (* I02 *)
  OR %M203                (* I03 *)
  OR %M204                (* I04 *)
  OR %M205                (* I05 *)
  OR %M212                (* I12 *)
  OR %M213                (* I13 *)
  OR %M214                (* I14 *)
  AND %M19                (* ARMED *)
  S %M20                  (* TRIGGERED *)
  // as ST:
  //   IF (I02 OR I03 OR I04 OR I05 OR I12 OR I13 OR I14) AND ARMED THEN TRIGGERED := TRUE; END_IF;

// Rung 70: START TIMER BEFORE CALLING SECURITY FIRM
  BLK %TM6                (* TRIG_TM *)
  LD %M20                 (* TRIGGERED *)
  IN
  OUT_BLK
  LD Q
  ANDN %M27               (* SS_TESTING_MODE *)
  ST %M237                (* Q13 *)
  END_BLK
  // as ST:
  //   TRIG_TM(IN := TRIGGERED);
  //   Q13 := TRIG_TM.Q AND NOT SS_TESTING_MODE;

// Rung 71: CONFIGURE BUZZER LOUDNESS
  LD %M20                 (* TRIGGERED *)
  [ %PWM1.R := ( %RTC0.SECONDS - %RTC0.SECONDS / 10 ) * 10 ](* BUZZER, RTC, RTC *)
  ST %M225                (* PWM1_IN *)
  // as ST:
  //   IF TRIGGERED THEN BUZZER.R := ( RTC.SECONDS - RTC.SECONDS / 10 ) * 10; END_IF;
  //   PWM1_IN := TRIGGERED;

Subroutine TEMP_REGULATOR
  (* SectionNumber=7, Number=5 *)

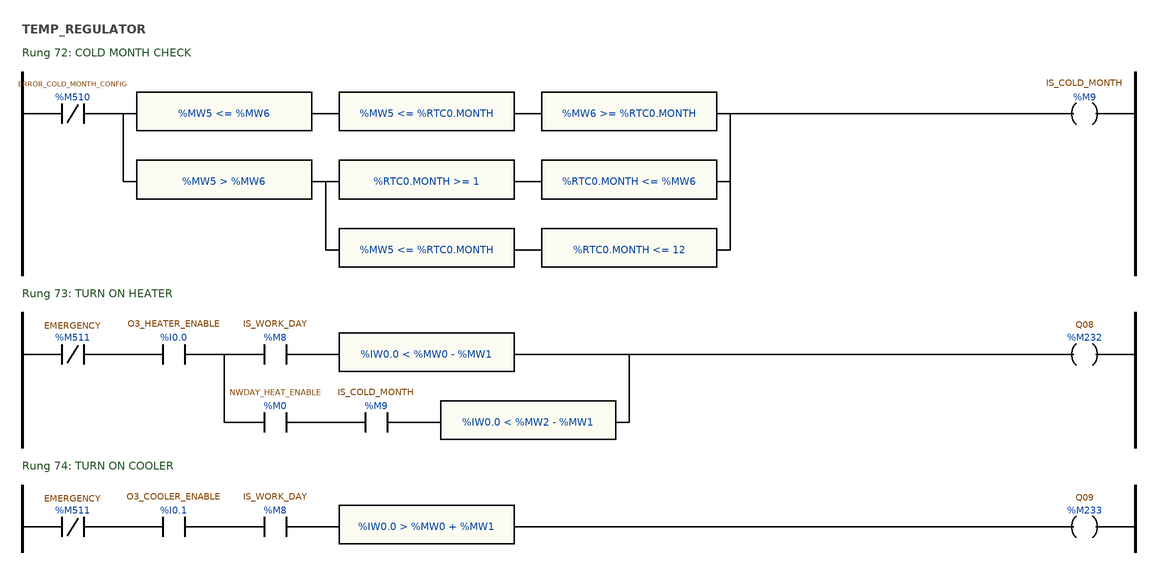

// Rung 72: COLD MONTH CHECK
  LDN %M510               (* ERROR_COLD_MONTH_CONFIG *)
  AND( [ %MW5 <= %MW6 ]   (* COLD_MONTH_START, COLD_MONTH_END *)
  AND [ %MW5 <= %RTC0.MONTH ](* COLD_MONTH_START, RTC *)
  AND [ %MW6 >= %RTC0.MONTH ](* COLD_MONTH_END, RTC *)
  OR( [ %MW5 > %MW6 ]     (* COLD_MONTH_START, COLD_MONTH_END *)
  AND( [ %RTC0.MONTH >= 1 ](* RTC *)
  AND [ %RTC0.MONTH <= %MW6 ](* RTC, COLD_MONTH_END *)
  OR( [ %MW5 <= %RTC0.MONTH ](* COLD_MONTH_START, RTC *)
  AND [ %RTC0.MONTH <= 12 ](* RTC *)
  )
  )
  )
  )
  ST %M9                  (* IS_COLD_MONTH *)
  // as ST:
  //   IS_COLD_MONTH := NOT ERROR_COLD_MONTH_CONFIG AND (COLD_MONTH_START <= COLD_MONTH_END AND COLD_MONTH_START <= RTC.MONTH AND COLD_MONTH_END >= RTC.MONTH OR COLD_MONTH_START > COLD_MONTH_END AND (RTC.MONTH >= 1 AND RTC.MONTH <= COLD_MONTH_END OR COLD_MONTH_START <= RTC.MONTH AND RTC.MONTH <= 12));

// Rung 73: TURN ON HEATER
  LDN %M511               (* EMERGENCY *)
  AND %I0.0               (* O3_HEATER_ENABLE *)
  AND( %M8                (* IS_WORK_DAY *)
  AND [ %IW0.0 < %MW0 - %MW1 ](* MEASURED_TEMP, DESIRED_TEMP, TOLERANCE_TEMP *)
  OR( %M0                 (* NWDAY_HEAT_ENABLE *)
  AND %M9                 (* IS_COLD_MONTH *)
  AND [ %IW0.0 < %MW2 - %MW1 ](* MEASURED_TEMP, NWDAY_DESIRED_TEMP, TOLERANCE_TEMP *)
  )
  )
  ST %M232                (* Q08 *)
  // as ST:
  //   Q08 := NOT EMERGENCY AND O3_HEATER_ENABLE AND (IS_WORK_DAY AND MEASURED_TEMP < DESIRED_TEMP - TOLERANCE_TEMP OR NWDAY_HEAT_ENABLE AND IS_COLD_MONTH AND MEASURED_TEMP < NWDAY_DESIRED_TEMP - TOLERANCE_TEMP);

// Rung 74: TURN ON COOLER
  LDN %M511               (* EMERGENCY *)
  AND %I0.1               (* O3_COOLER_ENABLE *)
  AND %M8                 (* IS_WORK_DAY *)
  AND [ %IW0.0 > %MW0 + %MW1 ](* MEASURED_TEMP, DESIRED_TEMP, TOLERANCE_TEMP *)
  ST %M233                (* Q09 *)
  // as ST:
  //   Q09 := NOT EMERGENCY AND O3_COOLER_ENABLE AND IS_WORK_DAY AND MEASURED_TEMP > DESIRED_TEMP + TOLERANCE_TEMP;

Subroutine RFID1_LOBBY
  (* SectionNumber=8, Number=11 *)

// Rung 75: REQUEST VALUE IS DEFAULT
  LD %M100                (* RFID1_REQUEST *)
  AND [ %MW100 = 0 ]      (* RFID1_REQ_START *)
  AND [ %MW101 = 0 ]      (* RFID1_REQ_MID *)
  AND [ %MW102 = 0 ]      (* RFID1_REQ_END *)
  S %M103                 (* RFID1_DENIED *)
  // as ST:
  //   IF RFID1_REQUEST AND RFID1_REQ_START = 0 AND RFID1_REQ_MID = 0 AND RFID1_REQ_END = 0 THEN RFID1_DENIED := TRUE; END_IF;

// Rung 76: RESPONSE BEFORE REQUEST
  LDN %M100               (* RFID1_REQUEST *)
  AND %M101               (* RFID1_RESPONSE *)
  S %M103                 (* RFID1_DENIED *)
  // as ST:
  //   IF NOT RFID1_REQUEST AND RFID1_RESPONSE THEN RFID1_DENIED := TRUE; END_IF;

// Rung 77: REQUEST CONDITION MET
  LDN %M103               (* RFID1_DENIED *)
  AND %M100               (* RFID1_REQUEST *)
  AND %M101               (* RFID1_RESPONSE *)
  AND [ %MW100 = %MW103 ] (* RFID1_REQ_START, RFID1_RESP_START *)
  AND [ %MW101 = %MW104 ] (* RFID1_REQ_MID, RFID1_RESP_MID *)
  AND [ %MW102 = %MW105 ] (* RFID1_REQ_END, RFID1_RESP_END *)
  S %M102                 (* RFID1_ACCEPT *)
  // as ST:
  //   IF NOT RFID1_DENIED AND RFID1_REQUEST AND RFID1_RESPONSE AND RFID1_REQ_START = RFID1_RESP_START AND RFID1_REQ_MID = RFID1_RESP_MID AND RFID1_REQ_END = RFID1_RESP_END THEN RFID1_ACCEPT := TRUE; END_IF;

// Rung 78: REQUEST CONDITION NOT MET
  LDN %M103               (* RFID1_DENIED *)
  AND %M100               (* RFID1_REQUEST *)
  AND %M101               (* RFID1_RESPONSE *)
  ANDN %M102              (* RFID1_ACCEPT *)
  S %M103                 (* RFID1_DENIED *)
  // as ST:
  //   IF NOT RFID1_DENIED AND RFID1_REQUEST AND RFID1_RESPONSE AND NOT RFID1_ACCEPT THEN RFID1_DENIED := TRUE; END_IF;

// Rung 79: OPEN LOCK FOR 3 SECONDS
  BLK %TM0                (* RFID1_TM *)
  LD %M102                (* RFID1_ACCEPT *)
  IN
  OUT_BLK
  LD Q
  S %M226                 (* Q02 *)
  END_BLK
  // as ST:
  //   RFID1_TM(IN := RFID1_ACCEPT);
  //   IF RFID1_TM.Q THEN Q02 := TRUE; END_IF;

// Rung 80: TIMER RAN OUT
  LD %M102                (* RFID1_ACCEPT *)
  ANDN %TM0.Q             (* RFID1_TM *)
  R %M102                 (* RFID1_ACCEPT *)
  R %M226                 (* Q02 *)
  // as ST:
  //   _t1 := RFID1_ACCEPT AND NOT RFID1_TM.Q;
  //   IF _t1 THEN RFID1_ACCEPT := FALSE; END_IF;
  //   IF _t1 THEN Q02 := FALSE; END_IF;

// Rung 81: RESTORE DEFAULT VALUES
  LDR %M102               (* RFID1_ACCEPT *)
  ORR %M103               (* RFID1_DENIED *)
  [ %MW100 := 0 ]         (* RFID1_REQ_START *)
  [ %MW101 := 0 ]         (* RFID1_REQ_MID *)
  [ %MW102 := 0 ]         (* RFID1_REQ_END *)
  [ %MW103 := 0 ]         (* RFID1_RESP_START *)
  [ %MW104 := 0 ]         (* RFID1_RESP_MID *)
  [ %MW105 := 0 ]         (* RFID1_RESP_END *)
  R %M100                 (* RFID1_REQUEST *)
  R %M101                 (* RFID1_RESPONSE *)
  // as ST:
  //   IF RISING(RFID1_ACCEPT) OR RISING(RFID1_DENIED) THEN RFID1_REQ_START := 0; END_IF;
  //   IF RISING(RFID1_ACCEPT) OR RISING(RFID1_DENIED) THEN RFID1_REQ_MID := 0; END_IF;
  //   IF RISING(RFID1_ACCEPT) OR RISING(RFID1_DENIED) THEN RFID1_REQ_END := 0; END_IF;
  //   IF RISING(RFID1_ACCEPT) OR RISING(RFID1_DENIED) THEN RFID1_RESP_START := 0; END_IF;
  //   IF RISING(RFID1_ACCEPT) OR RISING(RFID1_DENIED) THEN RFID1_RESP_MID := 0; END_IF;
  //   IF RISING(RFID1_ACCEPT) OR RISING(RFID1_DENIED) THEN RFID1_RESP_END := 0; END_IF;
  //   IF RISING(RFID1_ACCEPT) OR RISING(RFID1_DENIED) THEN RFID1_REQUEST := FALSE; END_IF;
  //   IF RISING(RFID1_ACCEPT) OR RISING(RFID1_DENIED) THEN RFID1_RESPONSE := FALSE; END_IF;

// Rung 82: RESTORE DENIED
  LDR %M103               (* RFID1_DENIED *)
  R %M103                 (* RFID1_DENIED *)
  // as ST:
  //   IF RISING(RFID1_DENIED) THEN RFID1_DENIED := FALSE; END_IF;

Subroutine RFID2_OFFICE1
  (* SectionNumber=9, Number=12 *)

// Rung 83: REQUEST VALUE IS DEFAULT
  LD %M106                (* RFID2_REQUEST *)
  AND [ %MW106 = 0 ]      (* RFID2_REQ_START *)
  AND [ %MW107 = 0 ]      (* RFID2_REQ_MID *)
  AND [ %MW108 = 0 ]      (* RFID2_REQ_END *)
  S %M109                 (* RFID2_DENIED *)
  // as ST:
  //   IF RFID2_REQUEST AND RFID2_REQ_START = 0 AND RFID2_REQ_MID = 0 AND RFID2_REQ_END = 0 THEN RFID2_DENIED := TRUE; END_IF;

// Rung 84: RESPONSE BEFORE REQUEST
  LDN %M106               (* RFID2_REQUEST *)
  AND %M107               (* RFID2_RESPONSE *)
  S %M109                 (* RFID2_DENIED *)
  // as ST:
  //   IF NOT RFID2_REQUEST AND RFID2_RESPONSE THEN RFID2_DENIED := TRUE; END_IF;

// Rung 85: REQUEST CONDITION MET
  LDN %M109               (* RFID2_DENIED *)
  AND %M106               (* RFID2_REQUEST *)
  AND %M107               (* RFID2_RESPONSE *)
  AND [ %MW106 = %MW109 ] (* RFID2_REQ_START, RFID2_RESP_START *)
  AND [ %MW107 = %MW110 ] (* RFID2_REQ_MID, RFID2_RESP_MID *)
  AND [ %MW108 = %MW111 ] (* RFID2_REQ_END, RFID2_RESP_END *)
  S %M108                 (* RFID2_ACCEPT *)
  // as ST:
  //   IF NOT RFID2_DENIED AND RFID2_REQUEST AND RFID2_RESPONSE AND RFID2_REQ_START = RFID2_RESP_START AND RFID2_REQ_MID = RFID2_RESP_MID AND RFID2_REQ_END = RFID2_RESP_END THEN RFID2_ACCEPT := TRUE; END_IF;

// Rung 86: REQUEST CONDITION NOT MET
  LDN %M109               (* RFID2_DENIED *)
  AND %M106               (* RFID2_REQUEST *)
  AND %M107               (* RFID2_RESPONSE *)
  ANDN %M108              (* RFID2_ACCEPT *)
  S %M109                 (* RFID2_DENIED *)
  // as ST:
  //   IF NOT RFID2_DENIED AND RFID2_REQUEST AND RFID2_RESPONSE AND NOT RFID2_ACCEPT THEN RFID2_DENIED := TRUE; END_IF;

// Rung 87: OPEN LOCK FOR 3 SECONDS
  BLK %TM1                (* RFID2_TM *)
  LD %M108                (* RFID2_ACCEPT *)
  IN
  OUT_BLK
  LD Q
  S %M227                 (* Q03 *)
  END_BLK
  // as ST:
  //   RFID2_TM(IN := RFID2_ACCEPT);
  //   IF RFID2_TM.Q THEN Q03 := TRUE; END_IF;

// Rung 88: TIMER RAN OUT
  LD %M108                (* RFID2_ACCEPT *)
  ANDN %TM1.Q             (* RFID2_TM *)
  R %M108                 (* RFID2_ACCEPT *)
  R %M227                 (* Q03 *)
  // as ST:
  //   _t1 := RFID2_ACCEPT AND NOT RFID2_TM.Q;
  //   IF _t1 THEN RFID2_ACCEPT := FALSE; END_IF;
  //   IF _t1 THEN Q03 := FALSE; END_IF;

// Rung 89: RESTORE DEFAULT VALUES
  LDR %M108               (* RFID2_ACCEPT *)
  ORR %M109               (* RFID2_DENIED *)
  [ %MW106 := 0 ]         (* RFID2_REQ_START *)
  [ %MW107 := 0 ]         (* RFID2_REQ_MID *)
  [ %MW108 := 0 ]         (* RFID2_REQ_END *)
  [ %MW109 := 0 ]         (* RFID2_RESP_START *)
  [ %MW110 := 0 ]         (* RFID2_RESP_MID *)
  [ %MW111 := 0 ]         (* RFID2_RESP_END *)
  R %M106                 (* RFID2_REQUEST *)
  R %M107                 (* RFID2_RESPONSE *)
  // as ST:
  //   IF RISING(RFID2_ACCEPT) OR RISING(RFID2_DENIED) THEN RFID2_REQ_START := 0; END_IF;
  //   IF RISING(RFID2_ACCEPT) OR RISING(RFID2_DENIED) THEN RFID2_REQ_MID := 0; END_IF;
  //   IF RISING(RFID2_ACCEPT) OR RISING(RFID2_DENIED) THEN RFID2_REQ_END := 0; END_IF;
  //   IF RISING(RFID2_ACCEPT) OR RISING(RFID2_DENIED) THEN RFID2_RESP_START := 0; END_IF;
  //   IF RISING(RFID2_ACCEPT) OR RISING(RFID2_DENIED) THEN RFID2_RESP_MID := 0; END_IF;
  //   IF RISING(RFID2_ACCEPT) OR RISING(RFID2_DENIED) THEN RFID2_RESP_END := 0; END_IF;
  //   IF RISING(RFID2_ACCEPT) OR RISING(RFID2_DENIED) THEN RFID2_REQUEST := FALSE; END_IF;
  //   IF RISING(RFID2_ACCEPT) OR RISING(RFID2_DENIED) THEN RFID2_RESPONSE := FALSE; END_IF;

// Rung 90: RESTORE DENIED
  LDR %M109               (* RFID2_DENIED *)
  R %M109                 (* RFID2_DENIED *)
  // as ST:
  //   IF RISING(RFID2_DENIED) THEN RFID2_DENIED := FALSE; END_IF;

Subroutine RFID3_OFFICE2
  (* SectionNumber=10, Number=13 *)

// Rung 91: REQUEST VALUE IS DEFAULT
  LD %M112                (* RFID3_REQUEST *)
  AND [ %MW112 = 0 ]      (* RFID3_REQ_START *)
  AND [ %MW113 = 0 ]      (* RFID3_REQ_MID *)
  AND [ %MW114 = 0 ]      (* RFID3_REQ_END *)
  S %M115                 (* RFID3_DENIED *)
  // as ST:
  //   IF RFID3_REQUEST AND RFID3_REQ_START = 0 AND RFID3_REQ_MID = 0 AND RFID3_REQ_END = 0 THEN RFID3_DENIED := TRUE; END_IF;

// Rung 92: RESPONSE BEFORE REQUEST
  LDN %M112               (* RFID3_REQUEST *)
  AND %M113               (* RFID3_RESPONSE *)
  S %M115                 (* RFID3_DENIED *)
  // as ST:
  //   IF NOT RFID3_REQUEST AND RFID3_RESPONSE THEN RFID3_DENIED := TRUE; END_IF;

// Rung 93: REQUEST CONDITION MET
  LDN %M115               (* RFID3_DENIED *)
  AND %M112               (* RFID3_REQUEST *)
  AND %M113               (* RFID3_RESPONSE *)
  AND [ %MW112 = %MW109 ] (* RFID3_REQ_START, RFID2_RESP_START *)
  AND [ %MW113 = %MW110 ] (* RFID3_REQ_MID, RFID2_RESP_MID *)
  AND [ %MW114 = %MW111 ] (* RFID3_REQ_END, RFID2_RESP_END *)
  S %M114                 (* RFID3_ACCEPT *)
  // as ST:
  //   IF NOT RFID3_DENIED AND RFID3_REQUEST AND RFID3_RESPONSE AND RFID3_REQ_START = RFID2_RESP_START AND RFID3_REQ_MID = RFID2_RESP_MID AND RFID3_REQ_END = RFID2_RESP_END THEN RFID3_ACCEPT := TRUE; END_IF;

// Rung 94: REQUEST CONDITION NOT MET
  LDN %M115               (* RFID3_DENIED *)
  AND %M112               (* RFID3_REQUEST *)
  AND %M113               (* RFID3_RESPONSE *)
  ANDN %M114              (* RFID3_ACCEPT *)
  S %M115                 (* RFID3_DENIED *)
  // as ST:
  //   IF NOT RFID3_DENIED AND RFID3_REQUEST AND RFID3_RESPONSE AND NOT RFID3_ACCEPT THEN RFID3_DENIED := TRUE; END_IF;

// Rung 95: OPEN LOCK FOR 3 SECONDS
  BLK %TM2                (* RFID3_TM *)
  LD %M108                (* RFID2_ACCEPT *)
  IN
  OUT_BLK
  LD Q
  S %M228                 (* Q04 *)
  END_BLK
  // as ST:
  //   RFID3_TM(IN := RFID2_ACCEPT);
  //   IF RFID3_TM.Q THEN Q04 := TRUE; END_IF;

// Rung 96: TIMER RAN OUT
  LD %M114                (* RFID3_ACCEPT *)
  ANDN %TM2.Q             (* RFID3_TM *)
  R %M114                 (* RFID3_ACCEPT *)
  R %M228                 (* Q04 *)
  // as ST:
  //   _t1 := RFID3_ACCEPT AND NOT RFID3_TM.Q;
  //   IF _t1 THEN RFID3_ACCEPT := FALSE; END_IF;
  //   IF _t1 THEN Q04 := FALSE; END_IF;

// Rung 97: RESTORE DEFAULT VALUES
  LDR %M114               (* RFID3_ACCEPT *)
  ORR %M115               (* RFID3_DENIED *)
  [ %MW112 := 0 ]         (* RFID3_REQ_START *)
  [ %MW113 := 0 ]         (* RFID3_REQ_MID *)
  [ %MW114 := 0 ]         (* RFID3_REQ_END *)
  [ %MW115 := 0 ]         (* RFID3_RESP_START *)
  [ %MW116 := 0 ]         (* RFID3_RESP_MID *)
  [ %MW117 := 0 ]         (* RFID3_RESP_END *)
  R %M112                 (* RFID3_REQUEST *)
  R %M113                 (* RFID3_RESPONSE *)
  // as ST:
  //   IF RISING(RFID3_ACCEPT) OR RISING(RFID3_DENIED) THEN RFID3_REQ_START := 0; END_IF;
  //   IF RISING(RFID3_ACCEPT) OR RISING(RFID3_DENIED) THEN RFID3_REQ_MID := 0; END_IF;
  //   IF RISING(RFID3_ACCEPT) OR RISING(RFID3_DENIED) THEN RFID3_REQ_END := 0; END_IF;
  //   IF RISING(RFID3_ACCEPT) OR RISING(RFID3_DENIED) THEN RFID3_RESP_START := 0; END_IF;
  //   IF RISING(RFID3_ACCEPT) OR RISING(RFID3_DENIED) THEN RFID3_RESP_MID := 0; END_IF;
  //   IF RISING(RFID3_ACCEPT) OR RISING(RFID3_DENIED) THEN RFID3_RESP_END := 0; END_IF;
  //   IF RISING(RFID3_ACCEPT) OR RISING(RFID3_DENIED) THEN RFID3_REQUEST := FALSE; END_IF;
  //   IF RISING(RFID3_ACCEPT) OR RISING(RFID3_DENIED) THEN RFID3_RESPONSE := FALSE; END_IF;

// Rung 98: RESTORE DENIED
  LDR %M115               (* RFID3_DENIED *)
  R %M115                 (* RFID3_DENIED *)
  // as ST:
  //   IF RISING(RFID3_DENIED) THEN RFID3_DENIED := FALSE; END_IF;

Subroutine RFID4_OFFICE3
  (* SectionNumber=11, Number=14 *)

// Rung 99: REQUEST VALUE IS DEFAULT
  LD %M118                (* RFID4_REQUEST *)
  AND [ %MW118 = 0 ]      (* RFID4_REQ_START *)
  AND [ %MW119 = 0 ]      (* RFID4_REQ_MID *)
  AND [ %MW120 = 0 ]      (* RFID4_REQ_END *)
  S %M121                 (* RFID4_DENIED *)
  // as ST:
  //   IF RFID4_REQUEST AND RFID4_REQ_START = 0 AND RFID4_REQ_MID = 0 AND RFID4_REQ_END = 0 THEN RFID4_DENIED := TRUE; END_IF;

// Rung 100: RESPONSE BEFORE REQUEST
  LDN %M118               (* RFID4_REQUEST *)
  AND %M119               (* RFID4_RESPONSE *)
  S %M121                 (* RFID4_DENIED *)
  // as ST:
  //   IF NOT RFID4_REQUEST AND RFID4_RESPONSE THEN RFID4_DENIED := TRUE; END_IF;

// Rung 101: REQUEST CONDITION MET
  LDN %M121               (* RFID4_DENIED *)
  AND %M118               (* RFID4_REQUEST *)
  AND %M119               (* RFID4_RESPONSE *)
  AND [ %MW118 = %MW109 ] (* RFID4_REQ_START, RFID2_RESP_START *)
  AND [ %MW119 = %MW110 ] (* RFID4_REQ_MID, RFID2_RESP_MID *)
  AND [ %MW120 = %MW111 ] (* RFID4_REQ_END, RFID2_RESP_END *)
  S %M120                 (* RFID4_ACCEPT *)
  // as ST:
  //   IF NOT RFID4_DENIED AND RFID4_REQUEST AND RFID4_RESPONSE AND RFID4_REQ_START = RFID2_RESP_START AND RFID4_REQ_MID = RFID2_RESP_MID AND RFID4_REQ_END = RFID2_RESP_END THEN RFID4_ACCEPT := TRUE; END_IF;

// Rung 102: REQUEST CONDITION NOT MET
  LDN %M121               (* RFID4_DENIED *)
  AND %M118               (* RFID4_REQUEST *)
  AND %M119               (* RFID4_RESPONSE *)
  ANDN %M120              (* RFID4_ACCEPT *)
  S %M121                 (* RFID4_DENIED *)
  // as ST:
  //   IF NOT RFID4_DENIED AND RFID4_REQUEST AND RFID4_RESPONSE AND NOT RFID4_ACCEPT THEN RFID4_DENIED := TRUE; END_IF;

// Rung 103: OPEN LOCK FOR 3 SECONDS
  BLK %TM3                (* RFID4_TM *)
  LD %M120                (* RFID4_ACCEPT *)
  IN
  OUT_BLK
  LD Q
  S %M229                 (* Q05 *)
  END_BLK
  // as ST:
  //   RFID4_TM(IN := RFID4_ACCEPT);
  //   IF RFID4_TM.Q THEN Q05 := TRUE; END_IF;

// Rung 104: TIMER RAN OUT
  LD %M120                (* RFID4_ACCEPT *)
  ANDN %TM3.Q             (* RFID4_TM *)
  R %M120                 (* RFID4_ACCEPT *)
  R %M229                 (* Q05 *)
  // as ST:
  //   _t1 := RFID4_ACCEPT AND NOT RFID4_TM.Q;
  //   IF _t1 THEN RFID4_ACCEPT := FALSE; END_IF;
  //   IF _t1 THEN Q05 := FALSE; END_IF;

// Rung 105: RESTORE DEFAULT VALUES
  LDR %M120               (* RFID4_ACCEPT *)
  ORR %M121               (* RFID4_DENIED *)
  [ %MW118 := 0 ]         (* RFID4_REQ_START *)
  [ %MW119 := 0 ]         (* RFID4_REQ_MID *)
  [ %MW120 := 0 ]         (* RFID4_REQ_END *)
  [ %MW121 := 0 ]         (* RFID4_RESP_START *)
  [ %MW122 := 0 ]         (* RFID4_RESP_MID *)
  [ %MW123 := 0 ]         (* RFID4_RESP_END *)
  R %M118                 (* RFID4_REQUEST *)
  R %M119                 (* RFID4_RESPONSE *)
  // as ST:
  //   IF RISING(RFID4_ACCEPT) OR RISING(RFID4_DENIED) THEN RFID4_REQ_START := 0; END_IF;
  //   IF RISING(RFID4_ACCEPT) OR RISING(RFID4_DENIED) THEN RFID4_REQ_MID := 0; END_IF;
  //   IF RISING(RFID4_ACCEPT) OR RISING(RFID4_DENIED) THEN RFID4_REQ_END := 0; END_IF;
  //   IF RISING(RFID4_ACCEPT) OR RISING(RFID4_DENIED) THEN RFID4_RESP_START := 0; END_IF;
  //   IF RISING(RFID4_ACCEPT) OR RISING(RFID4_DENIED) THEN RFID4_RESP_MID := 0; END_IF;
  //   IF RISING(RFID4_ACCEPT) OR RISING(RFID4_DENIED) THEN RFID4_RESP_END := 0; END_IF;
  //   IF RISING(RFID4_ACCEPT) OR RISING(RFID4_DENIED) THEN RFID4_REQUEST := FALSE; END_IF;
  //   IF RISING(RFID4_ACCEPT) OR RISING(RFID4_DENIED) THEN RFID4_RESPONSE := FALSE; END_IF;

// Rung 106: RESTORE DENIED
  LDR %M121               (* RFID4_DENIED *)
  R %M121                 (* RFID4_DENIED *)
  // as ST:
  //   IF RISING(RFID4_DENIED) THEN RFID4_DENIED := FALSE; END_IF;

Subroutine RFID5_PGATE
  (* SectionNumber=12, Number=15 *)

// Rung 107: REQEST VALUE IS DEFAULT
  LD %M124                (* RFID5_REQUEST *)
  AND [ %MW124 = 0 ]      (* RFID5_REQ_START *)
  AND [ %MW125 = 0 ]      (* RFID5_REQ_MID *)
  AND [ %MW126 = 0 ]      (* RFID5_REQ_END *)
  S %M127                 (* RFID5_DENIED *)
  // as ST:
  //   IF RFID5_REQUEST AND RFID5_REQ_START = 0 AND RFID5_REQ_MID = 0 AND RFID5_REQ_END = 0 THEN RFID5_DENIED := TRUE; END_IF;

// Rung 108: RESPONSE BEFORE REQUEST
  LDN %M124               (* RFID5_REQUEST *)
  AND %M125               (* RFID5_RESPONSE *)
  S %M127                 (* RFID5_DENIED *)
  // as ST:
  //   IF NOT RFID5_REQUEST AND RFID5_RESPONSE THEN RFID5_DENIED := TRUE; END_IF;

// Rung 109: REQUEST CONDITION MET
  LDN %M127               (* RFID5_DENIED *)
  AND %M124               (* RFID5_REQUEST *)
  AND %M125               (* RFID5_RESPONSE *)
  AND [ %MW124 = %MW127 ] (* RFID5_REQ_START, RFID5_RESP_START *)
  AND [ %MW125 = %MW128 ] (* RFID5_REQ_MID, RFID5_RESP_MID *)
  AND [ %MW126 = %MW129 ] (* RFID5_REQ_END, RFID5_RESP_END *)
  S %M126                 (* PGATE_ACCEPT *)
  // as ST:
  //   IF NOT RFID5_DENIED AND RFID5_REQUEST AND RFID5_RESPONSE AND RFID5_REQ_START = RFID5_RESP_START AND RFID5_REQ_MID = RFID5_RESP_MID AND RFID5_REQ_END = RFID5_RESP_END THEN PGATE_ACCEPT := TRUE; END_IF;

// Rung 110: REQUEST CONDITION NOT MET
  LDN %M127               (* RFID5_DENIED *)
  AND %M124               (* RFID5_REQUEST *)
  AND %M125               (* RFID5_RESPONSE *)
  ANDN %M126              (* PGATE_ACCEPT *)
  S %M127                 (* RFID5_DENIED *)
  // as ST:
  //   IF NOT RFID5_DENIED AND RFID5_REQUEST AND RFID5_RESPONSE AND NOT PGATE_ACCEPT THEN RFID5_DENIED := TRUE; END_IF;

// Rung 111: START OUTSIDE PARKING CYCLE
  LDR %M126               (* PGATE_ACCEPT *)
  S %M14                  (* OUTSIDE_PCYCLE *)
  // as ST:
  //   IF RISING(PGATE_ACCEPT) THEN OUTSIDE_PCYCLE := TRUE; END_IF;

// Rung 112: RESTORE DEFAULT VALUES
  LDR %M126               (* PGATE_ACCEPT *)
  ORR %M127               (* RFID5_DENIED *)
  [ %MW124 := 0 ]         (* RFID5_REQ_START *)
  [ %MW125 := 0 ]         (* RFID5_REQ_MID *)
  [ %MW126 := 0 ]         (* RFID5_REQ_END *)
  [ %MW127 := 0 ]         (* RFID5_RESP_START *)
  [ %MW128 := 0 ]         (* RFID5_RESP_MID *)
  [ %MW129 := 0 ]         (* RFID5_RESP_END *)
  R %M124                 (* RFID5_REQUEST *)
  R %M125                 (* RFID5_RESPONSE *)
  // as ST:
  //   IF RISING(PGATE_ACCEPT) OR RISING(RFID5_DENIED) THEN RFID5_REQ_START := 0; END_IF;
  //   IF RISING(PGATE_ACCEPT) OR RISING(RFID5_DENIED) THEN RFID5_REQ_MID := 0; END_IF;
  //   IF RISING(PGATE_ACCEPT) OR RISING(RFID5_DENIED) THEN RFID5_REQ_END := 0; END_IF;
  //   IF RISING(PGATE_ACCEPT) OR RISING(RFID5_DENIED) THEN RFID5_RESP_START := 0; END_IF;
  //   IF RISING(PGATE_ACCEPT) OR RISING(RFID5_DENIED) THEN RFID5_RESP_MID := 0; END_IF;
  //   IF RISING(PGATE_ACCEPT) OR RISING(RFID5_DENIED) THEN RFID5_RESP_END := 0; END_IF;
  //   IF RISING(PGATE_ACCEPT) OR RISING(RFID5_DENIED) THEN RFID5_REQUEST := FALSE; END_IF;
  //   IF RISING(PGATE_ACCEPT) OR RISING(RFID5_DENIED) THEN RFID5_RESPONSE := FALSE; END_IF;

// Rung 113: RESTORE DENIED
  LDR %M127               (* RFID5_DENIED *)
  R %M127                 (* RFID5_DENIED *)
  // as ST:
  //   IF RISING(RFID5_DENIED) THEN RFID5_DENIED := FALSE; END_IF;

Subroutine PGATE_LOGIC
  (* SectionNumber=13, Number=16 *)

// Rung 114: PARKING LOT INDICATOR
// WHEN FULL OR EMERGENCY
  LD %M17                 (* PLOT_FULL *)
  OR %M511                (* EMERGENCY *)
  ST %M239                (* Q15 *)
  // as ST:
  //   Q15 := PLOT_FULL OR EMERGENCY;

// Rung 115: PGATE BUTTON PRESS
// FROM INSIDE PARKING LOT
  LDN %M511               (* EMERGENCY *)
  ANDN %M14               (* OUTSIDE_PCYCLE *)
  ANDR %I0.9              (* P_GATE_BTN *)
  S %M13                  (* INSIDE_PCYCLE *)
  S %M126                 (* PGATE_ACCEPT *)
  // as ST:
  //   IF NOT EMERGENCY AND NOT OUTSIDE_PCYCLE AND RISING(P_GATE_BTN) THEN INSIDE_PCYCLE := TRUE; END_IF;
  //   IF NOT EMERGENCY AND NOT OUTSIDE_PCYCLE AND RISING(P_GATE_BTN) THEN PGATE_ACCEPT := TRUE; END_IF;

// Rung 116: PGATE EMERGENCY BEHAVIOUR
  LDR %M511               (* EMERGENCY *)
  S %M128                 (* PGATE_FOPEN *)
  R %M129                 (* PGATE_FCLOSE *)
  // as ST:
  //   IF RISING(EMERGENCY) THEN PGATE_FOPEN := TRUE; END_IF;
  //   IF RISING(EMERGENCY) THEN PGATE_FCLOSE := FALSE; END_IF;

// Rung 117: PGATE OPEN OUTSIDE OCC
  LDN %M13                (* INSIDE_PCYCLE *)
  ANDN %M14               (* OUTSIDE_PCYCLE *)
  ANDN %M207              (* I07 *)
  ST %M498                (* WARNING_PGATE_OPENED *)
  // as ST:
  //   WARNING_PGATE_OPENED := NOT INSIDE_PCYCLE AND NOT OUTSIDE_PCYCLE AND NOT I07;

// Rung 118: FORCE RESET BITS
  LDR %M128               (* PGATE_FOPEN *)
  ANDN %M129              (* PGATE_FCLOSE *)
  OR(R %M129              (* PGATE_FCLOSE *)
  ANDN %M128              (* PGATE_FOPEN *)
  )
  R %M13                  (* INSIDE_PCYCLE *)
  R %M14                  (* OUTSIDE_PCYCLE *)
  R %M126                 (* PGATE_ACCEPT *)
  // as ST:
  //   IF RISING(PGATE_FOPEN) AND NOT PGATE_FCLOSE OR RISING(PGATE_FCLOSE) AND NOT PGATE_FOPEN THEN INSIDE_PCYCLE := FALSE; END_IF;
  //   IF RISING(PGATE_FOPEN) AND NOT PGATE_FCLOSE OR RISING(PGATE_FCLOSE) AND NOT PGATE_FOPEN THEN OUTSIDE_PCYCLE := FALSE; END_IF;
  //   IF RISING(PGATE_FOPEN) AND NOT PGATE_FCLOSE OR RISING(PGATE_FCLOSE) AND NOT PGATE_FOPEN THEN PGATE_ACCEPT := FALSE; END_IF;

// Rung 119: FORCE OPEN PARKING LOT GATE
// DOESN'T TRACK PASSING OBJECTS
  LD %M128                (* PGATE_FOPEN *)
  ANDN %M129              (* PGATE_FCLOSE *)
  ANDN %M206              (* I06 *)
  ST %M230                (* Q06 *)
  // as ST:
  //   Q06 := PGATE_FOPEN AND NOT PGATE_FCLOSE AND NOT I06;

// Rung 120: FORCE CLOSE PARKING LOT GATE
// DOESN'T TRACK PASSING OBJECTS
  LD %M129                (* PGATE_FCLOSE *)
  ANDN %M128              (* PGATE_FOPEN *)
  ANDN %M208              (* I08 *)
  ANDN %M207              (* I07 *)
  ST %M231                (* Q07 *)
  // as ST:
  //   Q07 := PGATE_FCLOSE AND NOT PGATE_FOPEN AND NOT I08 AND NOT I07;

// Rung 121: INDICATE FORCE OPEN AND CLOSE ERROR
  LD %M128                (* PGATE_FOPEN *)
  AND %M129               (* PGATE_FCLOSE *)
  ST %M506                (* ERROR_PGATE_FCLOPEN *)
  // as ST:
  //   ERROR_PGATE_FCLOPEN := PGATE_FOPEN AND PGATE_FCLOSE;

Subroutine PGATE_OCC  (* OPEN/CLOSE CYCLE FOR PARKING LOT GATE *)
  (* SectionNumber=14, Number=17 *)

// Rung 122: CHECK FOR CLOSED GATE
  LDR %I0.7               (* P_GATE_CLOSED *)
  MPS
  AND %M14                (* OUTSIDE_PCYCLE *)
  R %M14                  (* OUTSIDE_PCYCLE *)
  MRD
  AND %M13                (* INSIDE_PCYCLE *)
  R %M13                  (* INSIDE_PCYCLE *)
  MPP
  [ %MW11 := 0 ]          (* PGATE_PASSED_OBJECTS *)
  // as ST:
  //   IF RISING(P_GATE_CLOSED) AND OUTSIDE_PCYCLE THEN OUTSIDE_PCYCLE := FALSE; END_IF;
  //   IF RISING(P_GATE_CLOSED) AND INSIDE_PCYCLE THEN INSIDE_PCYCLE := FALSE; END_IF;
  //   IF RISING(P_GATE_CLOSED) THEN PGATE_PASSED_OBJECTS := 0; END_IF;

// Rung 123: OPEN PARKING DOOR
  LD %M126                (* PGATE_ACCEPT *)
  ANDN %I0.6              (* P_GATE_OPENED *)
  ST %M230                (* Q06 *)
  // as ST:
  //   Q06 := PGATE_ACCEPT AND NOT P_GATE_OPENED;

// Rung 124: START TIMER 20s
  BLK %TM4                (* PGATE_TM *)
  LD %M126                (* PGATE_ACCEPT *)
  AND %I0.6               (* P_GATE_OPENED *)
  IN
  END_BLK
  // as ST:
  //   PGATE_TM(IN := PGATE_ACCEPT AND P_GATE_OPENED);

// Rung 125: TIMER ENDED OR CAR PASSED
  LD %TM4.Q               (* PGATE_TM *)
  ORF %I0.8               (* P_GATE_OBJECT *)
  R %M126                 (* PGATE_ACCEPT *)
  // as ST:
  //   IF PGATE_TM.Q OR FALLING(P_GATE_OBJECT) THEN PGATE_ACCEPT := FALSE; END_IF;

// Rung 126: UPDATE PARKED CAR COUNT
  LDF %I0.8               (* P_GATE_OBJECT *)
  MPS
  AND %M14                (* OUTSIDE_PCYCLE *)
  [ %MW9 := %MW9 + 1 ]    (* PARKING_SPOTS_TAKEN, PARKING_SPOTS_TAKEN *)
  MRD
  AND %M13                (* INSIDE_PCYCLE *)
  [ %MW9 := %MW9 - 1 ]    (* PARKING_SPOTS_TAKEN, PARKING_SPOTS_TAKEN *)
  MPP
  [ %MW11 := %MW11 + 1 ]  (* PGATE_PASSED_OBJECTS, PGATE_PASSED_OBJECTS *)
  // as ST:
  //   IF FALLING(P_GATE_OBJECT) AND OUTSIDE_PCYCLE THEN PARKING_SPOTS_TAKEN := PARKING_SPOTS_TAKEN + 1; END_IF;
  //   IF FALLING(P_GATE_OBJECT) AND INSIDE_PCYCLE THEN PARKING_SPOTS_TAKEN := PARKING_SPOTS_TAKEN - 1; END_IF;
  //   IF FALLING(P_GATE_OBJECT) THEN PGATE_PASSED_OBJECTS := PGATE_PASSED_OBJECTS + 1; END_IF;

// Rung 127: PARKING SPOT MISCOUNT WARNING FLAG
  LDF %I0.8               (* P_GATE_OBJECT *)
  AND( [ %MW9 > %MW10 ]   (* PARKING_SPOTS_TAKEN, PARKING_SPOT_THCOUNT *)
  OR [ %MW9 < 0 ]         (* PARKING_SPOTS_TAKEN *)
  OR [ %MW11 > 1 ]        (* PGATE_PASSED_OBJECTS *)
  )
  S %M499                 (* WARNING_PSPOT_MISCOUNT *)
  // as ST:
  //   IF FALLING(P_GATE_OBJECT) AND (PARKING_SPOTS_TAKEN > PARKING_SPOT_THCOUNT OR PARKING_SPOTS_TAKEN < 0 OR PGATE_PASSED_OBJECTS > 1) THEN WARNING_PSPOT_MISCOUNT := TRUE; END_IF;

// Rung 128: PARKING LOT FULL OR OVER CAPACITY
  LDF %I0.8               (* P_GATE_OBJECT *)
  MPS
  AND [ %MW9 >= %MW8 ]    (* PARKING_SPOTS_TAKEN, PARKING_SPOT_COUNT *)
  S %M17                  (* PLOT_FULL *)
  MPP
  AND [ %MW9 < %MW8 ]     (* PARKING_SPOTS_TAKEN, PARKING_SPOT_COUNT *)
  R %M17                  (* PLOT_FULL *)
  // as ST:
  //   IF FALLING(P_GATE_OBJECT) AND PARKING_SPOTS_TAKEN >= PARKING_SPOT_COUNT THEN PLOT_FULL := TRUE; END_IF;
  //   IF FALLING(P_GATE_OBJECT) AND PARKING_SPOTS_TAKEN < PARKING_SPOT_COUNT THEN PLOT_FULL := FALSE; END_IF;

// Rung 129: CLOSE PARKING LOT GATE
  LDN %I0.7               (* P_GATE_CLOSED *)
  ANDN %M126              (* PGATE_ACCEPT *)
  ANDN %I0.8              (* P_GATE_OBJECT *)
  ST %M231                (* Q07 *)
  // as ST:
  //   Q07 := NOT P_GATE_CLOSED AND NOT PGATE_ACCEPT AND NOT P_GATE_OBJECT;

Subroutine SPECIAL_BEHAVIOR
  (* SectionNumber=15, Number=20 *)

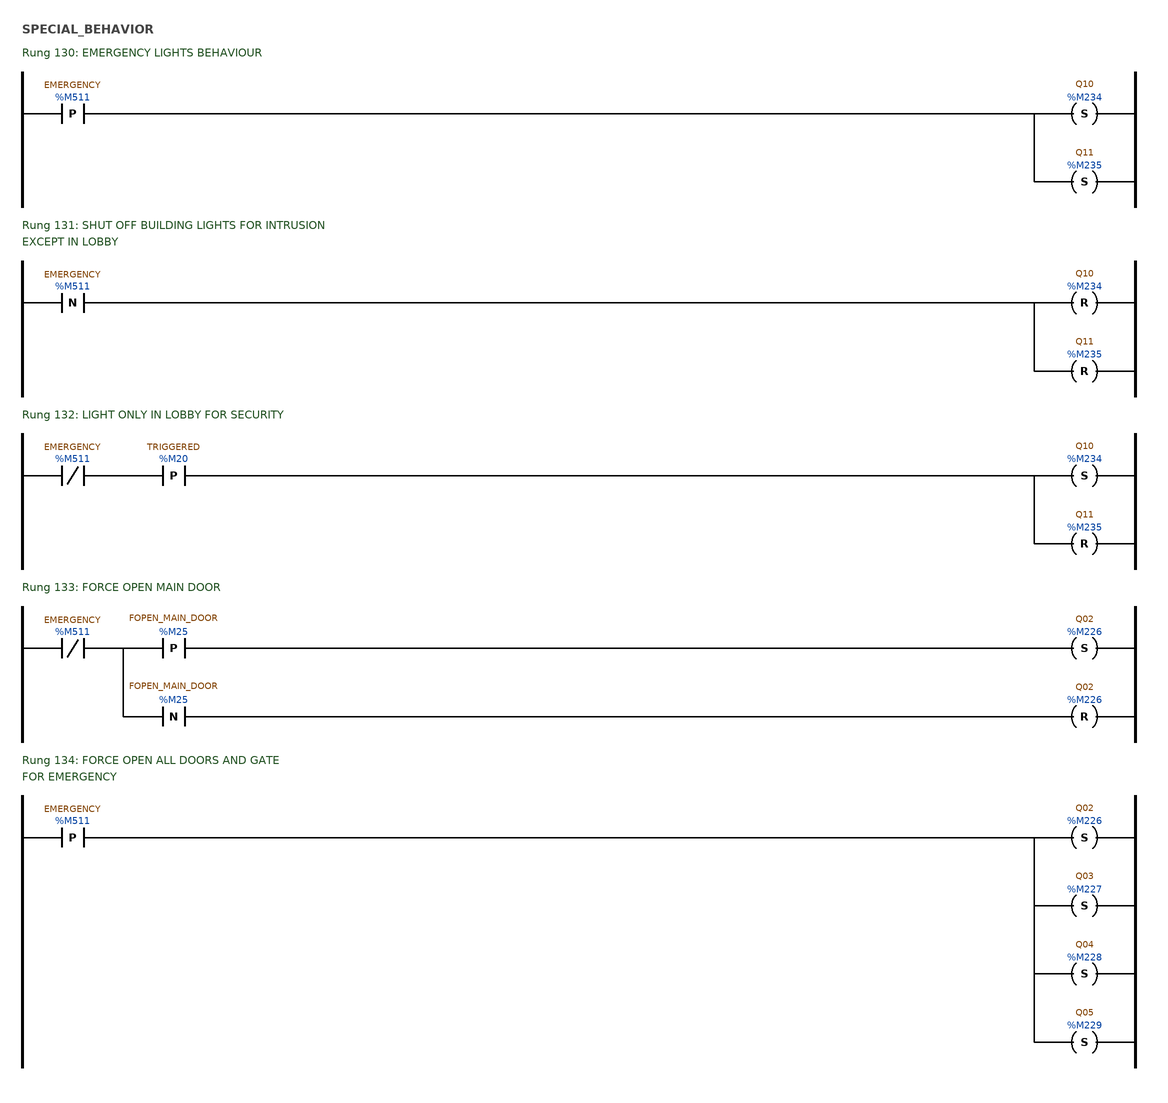

// Rung 130: EMERGENCY LIGHTS BEHAVIOUR
  LDR %M511               (* EMERGENCY *)
  S %M234                 (* Q10 *)
  S %M235                 (* Q11 *)
  // as ST:
  //   IF RISING(EMERGENCY) THEN Q10 := TRUE; END_IF;
  //   IF RISING(EMERGENCY) THEN Q11 := TRUE; END_IF;

// Rung 131: SHUT OFF BUILDING LIGHTS FOR INTRUSION
// EXCEPT IN LOBBY
  LDF %M511               (* EMERGENCY *)
  R %M234                 (* Q10 *)
  R %M235                 (* Q11 *)
  // as ST:
  //   IF FALLING(EMERGENCY) THEN Q10 := FALSE; END_IF;
  //   IF FALLING(EMERGENCY) THEN Q11 := FALSE; END_IF;

// Rung 132: LIGHT ONLY IN LOBBY FOR SECURITY
  LDN %M511               (* EMERGENCY *)
  ANDR %M20               (* TRIGGERED *)
  S %M234                 (* Q10 *)
  R %M235                 (* Q11 *)
  // as ST:
  //   IF NOT EMERGENCY AND RISING(TRIGGERED) THEN Q10 := TRUE; END_IF;
  //   IF NOT EMERGENCY AND RISING(TRIGGERED) THEN Q11 := FALSE; END_IF;

// Rung 133: FORCE OPEN MAIN DOOR
  LDN %M511               (* EMERGENCY *)
  MPS
  ANDR %M25               (* FOPEN_MAIN_DOOR *)
  S %M226                 (* Q02 *)
  MPP
  ANDF %M25               (* FOPEN_MAIN_DOOR *)
  R %M226                 (* Q02 *)
  // as ST:
  //   IF NOT EMERGENCY AND RISING(FOPEN_MAIN_DOOR) THEN Q02 := TRUE; END_IF;
  //   IF NOT EMERGENCY AND FALLING(FOPEN_MAIN_DOOR) THEN Q02 := FALSE; END_IF;

// Rung 134: FORCE OPEN ALL DOORS AND GATE
// FOR EMERGENCY
  LDR %M511               (* EMERGENCY *)
  S %M226                 (* Q02 *)
  S %M227                 (* Q03 *)
  S %M228                 (* Q04 *)
  S %M229                 (* Q05 *)
  // as ST:
  //   IF RISING(EMERGENCY) THEN Q02 := TRUE; END_IF;
  //   IF RISING(EMERGENCY) THEN Q03 := TRUE; END_IF;
  //   IF RISING(EMERGENCY) THEN Q04 := TRUE; END_IF;
  //   IF RISING(EMERGENCY) THEN Q05 := TRUE; END_IF;

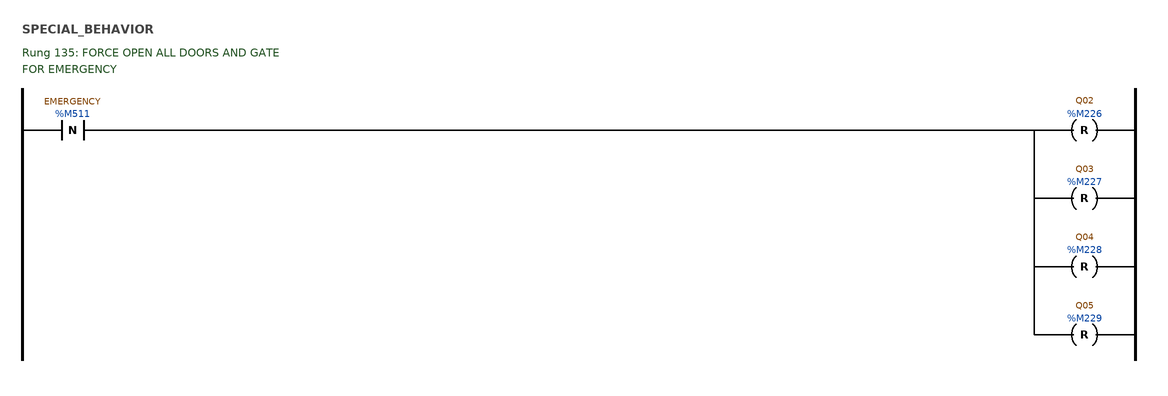

// Rung 135: FORCE OPEN ALL DOORS AND GATE
// FOR EMERGENCY
  LDF %M511               (* EMERGENCY *)
  R %M226                 (* Q02 *)
  R %M227                 (* Q03 *)
  R %M228                 (* Q04 *)
  R %M229                 (* Q05 *)
  // as ST:
  //   IF FALLING(EMERGENCY) THEN Q02 := FALSE; END_IF;
  //   IF FALLING(EMERGENCY) THEN Q03 := FALSE; END_IF;
  //   IF FALLING(EMERGENCY) THEN Q04 := FALSE; END_IF;
  //   IF FALLING(EMERGENCY) THEN Q05 := FALSE; END_IF;

Subroutine LIGHTS_LOBBY
  (* SectionNumber=16, Number=21 *)

// Rung 136: ENABLE BUTTON INPUT
  LDN %M28                (* AUTO_LIGHTS_L *)
  OR( %M28                (* AUTO_LIGHTS_L *)
  AND %M29                (* WDONLY_LIGHTS_L *)
  ANDN %M8                (* IS_WORK_DAY *)
  )
  ST %M30                 (* BTN_ENABLE_LIGHTS_L *)
  // as ST:
  //   BTN_ENABLE_LIGHTS_L := NOT AUTO_LIGHTS_L OR AUTO_LIGHTS_L AND WDONLY_LIGHTS_L AND NOT IS_WORK_DAY;

// Rung 137: MANUAL LIGHT OFF
  LDF %M30                (* BTN_ENABLE_LIGHTS_L *)
  R %M234                 (* Q10 *)
  // as ST:
  //   IF FALLING(BTN_ENABLE_LIGHTS_L) THEN Q10 := FALSE; END_IF;

// Rung 138: BUTTON LIGHTS ON
  LD %M30                 (* BTN_ENABLE_LIGHTS_L *)
  ANDR %M211              (* I11 *)
  ANDN %M234              (* Q10 *)
  S %M234                 (* Q10 *)
  S %M33                  (* CHANGED_LIGHTS_L *)
  // as ST:
  //   _t1 := BTN_ENABLE_LIGHTS_L AND RISING(I11) AND NOT Q10;
  //   IF _t1 THEN Q10 := TRUE; END_IF;
  //   IF _t1 THEN CHANGED_LIGHTS_L := TRUE; END_IF;

// Rung 139: BUTTON LIGHTS OFF
  LDN %M33                (* CHANGED_LIGHTS_L *)
  AND %M30                (* BTN_ENABLE_LIGHTS_L *)
  ANDR %M211              (* I11 *)
  AND %M234               (* Q10 *)
  R %M234                 (* Q10 *)
  // as ST:
  //   IF NOT CHANGED_LIGHTS_L AND BTN_ENABLE_LIGHTS_L AND RISING(I11) AND Q10 THEN Q10 := FALSE; END_IF;

// Rung 140: RESET CHANGED BIT
  LD %M33                 (* CHANGED_LIGHTS_L *)
  R %M33                  (* CHANGED_LIGHTS_L *)
  // as ST:
  //   IF CHANGED_LIGHTS_L THEN CHANGED_LIGHTS_L := FALSE; END_IF;

// Rung 141: SET MOVEMENT DETECTED BIT
  LD %M212                (* I12 *)
  AND %M32                (* AUTO_MODE_LIGHTS_L *)
  S %M34                  (* MOVEMENT_LIGHTS_L *)
  // as ST:
  //   IF I12 AND AUTO_MODE_LIGHTS_L THEN MOVEMENT_LIGHTS_L := TRUE; END_IF;

// Rung 142: AUTOMATIC MODES ON
// MOVEMENT OR KEEP ON
  LDN %M30                (* BTN_ENABLE_LIGHTS_L *)
  AND( %M34               (* MOVEMENT_LIGHTS_L *)
  ORN %M32                (* AUTO_MODE_LIGHTS_L *)
  )
  AND [ %MW201 <= %MW14 ] (* IW1, TRESHOLD_LIGHTS *)
  S %M234                 (* Q10 *)
  // as ST:
  //   IF NOT BTN_ENABLE_LIGHTS_L AND (MOVEMENT_LIGHTS_L OR NOT AUTO_MODE_LIGHTS_L) AND IW1 <= TRESHOLD_LIGHTS THEN Q10 := TRUE; END_IF;

// Rung 143: AUTOMATIC MODE 1 OFF
  BLK %TM8                (* LIGHT_TM_L *)
  LD %M34                 (* MOVEMENT_LIGHTS_L *)
  IN
  OUT_BLK
  LD Q
  R %M234                 (* Q10 *)
  R %M34                  (* MOVEMENT_LIGHTS_L *)
  END_BLK
  // as ST:
  //   LIGHT_TM_L(IN := MOVEMENT_LIGHTS_L);
  //   IF LIGHT_TM_L.Q THEN Q10 := FALSE; END_IF;
  //   IF LIGHT_TM_L.Q THEN MOVEMENT_LIGHTS_L := FALSE; END_IF;

// Rung 144: AUTOMATIC MODE 0 OFF
  LD %M234                (* Q10 *)
  ANDN %M32               (* AUTO_MODE_LIGHTS_L *)
  AND [ %MW201 > %MW14 + %MW15 ](* IW1, TRESHOLD_LIGHTS, TOLERANCE_LIGHTS *)
  R %M234                 (* Q10 *)
  // as ST:
  //   IF Q10 AND NOT AUTO_MODE_LIGHTS_L AND IW1 > TRESHOLD_LIGHTS + TOLERANCE_LIGHTS THEN Q10 := FALSE; END_IF;

Subroutine LIGHTS_BUILDING
  (* SectionNumber=17, Number=22 *)

// Rung 145: ENABLE BUTTON INPUT
  LDN %M35                (* AUTO_LIGHTS_B *)
  OR( %M35                (* AUTO_LIGHTS_B *)
  AND %M36                (* WDONLY_LIGHTS_B *)
  ANDN %M8                (* IS_WORK_DAY *)
  )
  ST %M37                 (* BTN_ENABLE_LIGHTS_B *)
  // as ST:
  //   BTN_ENABLE_LIGHTS_B := NOT AUTO_LIGHTS_B OR AUTO_LIGHTS_B AND WDONLY_LIGHTS_B AND NOT IS_WORK_DAY;

// Rung 146: MANUAL LIGHT OFF
  LDF %M37                (* BTN_ENABLE_LIGHTS_B *)
  R %M235                 (* Q11 *)
  // as ST:
  //   IF FALLING(BTN_ENABLE_LIGHTS_B) THEN Q11 := FALSE; END_IF;

// Rung 147: BUTTON LIGHTS ON
  LD %M37                 (* BTN_ENABLE_LIGHTS_B *)
  ANDR %M211              (* I11 *)
  ANDN %M235              (* Q11 *)
  S %M235                 (* Q11 *)
  S %M41                  (* MOVEMENT_LIGHTS_B *)
  // as ST:
  //   _t1 := BTN_ENABLE_LIGHTS_B AND RISING(I11) AND NOT Q11;
  //   IF _t1 THEN Q11 := TRUE; END_IF;
  //   IF _t1 THEN MOVEMENT_LIGHTS_B := TRUE; END_IF;

// Rung 148: BUTTON LIGHTS OFF
  LDN %M40                (* CHANGED_LIGHTS_B *)
  AND %M37                (* BTN_ENABLE_LIGHTS_B *)
  ANDR %M211              (* I11 *)
  AND %M235               (* Q11 *)
  R %M235                 (* Q11 *)
  // as ST:
  //   IF NOT CHANGED_LIGHTS_B AND BTN_ENABLE_LIGHTS_B AND RISING(I11) AND Q11 THEN Q11 := FALSE; END_IF;

// Rung 149: RESET CHANGED BIT
  LD %M40                 (* CHANGED_LIGHTS_B *)
  R %M40                  (* CHANGED_LIGHTS_B *)
  // as ST:
  //   IF CHANGED_LIGHTS_B THEN CHANGED_LIGHTS_B := FALSE; END_IF;

// Rung 150: SET MOVEMENT DETECTED BIT
  LD %M212                (* I12 *)
  AND %M39                (* AUTO_MODE_LIGHTS_B *)
  S %M41                  (* MOVEMENT_LIGHTS_B *)
  // as ST:
  //   IF I12 AND AUTO_MODE_LIGHTS_B THEN MOVEMENT_LIGHTS_B := TRUE; END_IF;

// Rung 151: AUTOMATIC MODES ON
// MOVEMENT OR KEEP ON
  LDN %M37                (* BTN_ENABLE_LIGHTS_B *)
  AND( %M41               (* MOVEMENT_LIGHTS_B *)
  ORN %M39                (* AUTO_MODE_LIGHTS_B *)
  )
  AND [ %MW201 <= %MW14 ] (* IW1, TRESHOLD_LIGHTS *)
  S %M235                 (* Q11 *)
  // as ST:
  //   IF NOT BTN_ENABLE_LIGHTS_B AND (MOVEMENT_LIGHTS_B OR NOT AUTO_MODE_LIGHTS_B) AND IW1 <= TRESHOLD_LIGHTS THEN Q11 := TRUE; END_IF;

// Rung 152: AUTOMATIC MODE 1 OFF
  BLK %TM9                (* LIGHT_TM_B *)
  LD %M41                 (* MOVEMENT_LIGHTS_B *)
  IN
  OUT_BLK
  LD Q
  R %M235                 (* Q11 *)
  R %M41                  (* MOVEMENT_LIGHTS_B *)
  END_BLK
  // as ST:
  //   LIGHT_TM_B(IN := MOVEMENT_LIGHTS_B);
  //   IF LIGHT_TM_B.Q THEN Q11 := FALSE; END_IF;
  //   IF LIGHT_TM_B.Q THEN MOVEMENT_LIGHTS_B := FALSE; END_IF;

// Rung 153: AUTOMATIC MODE 0 OFF
  LD %M235                (* Q11 *)
  ANDN %M39               (* AUTO_MODE_LIGHTS_B *)
  AND [ %MW201 > %MW14 + %MW15 ](* IW1, TRESHOLD_LIGHTS, TOLERANCE_LIGHTS *)
  R %M235                 (* Q11 *)
  // as ST:
  //   IF Q11 AND NOT AUTO_MODE_LIGHTS_B AND IW1 > TRESHOLD_LIGHTS + TOLERANCE_LIGHTS THEN Q11 := FALSE; END_IF;

Subroutine RECORD_OUTPUTS
  (* SectionNumber=18, Number=63 *)

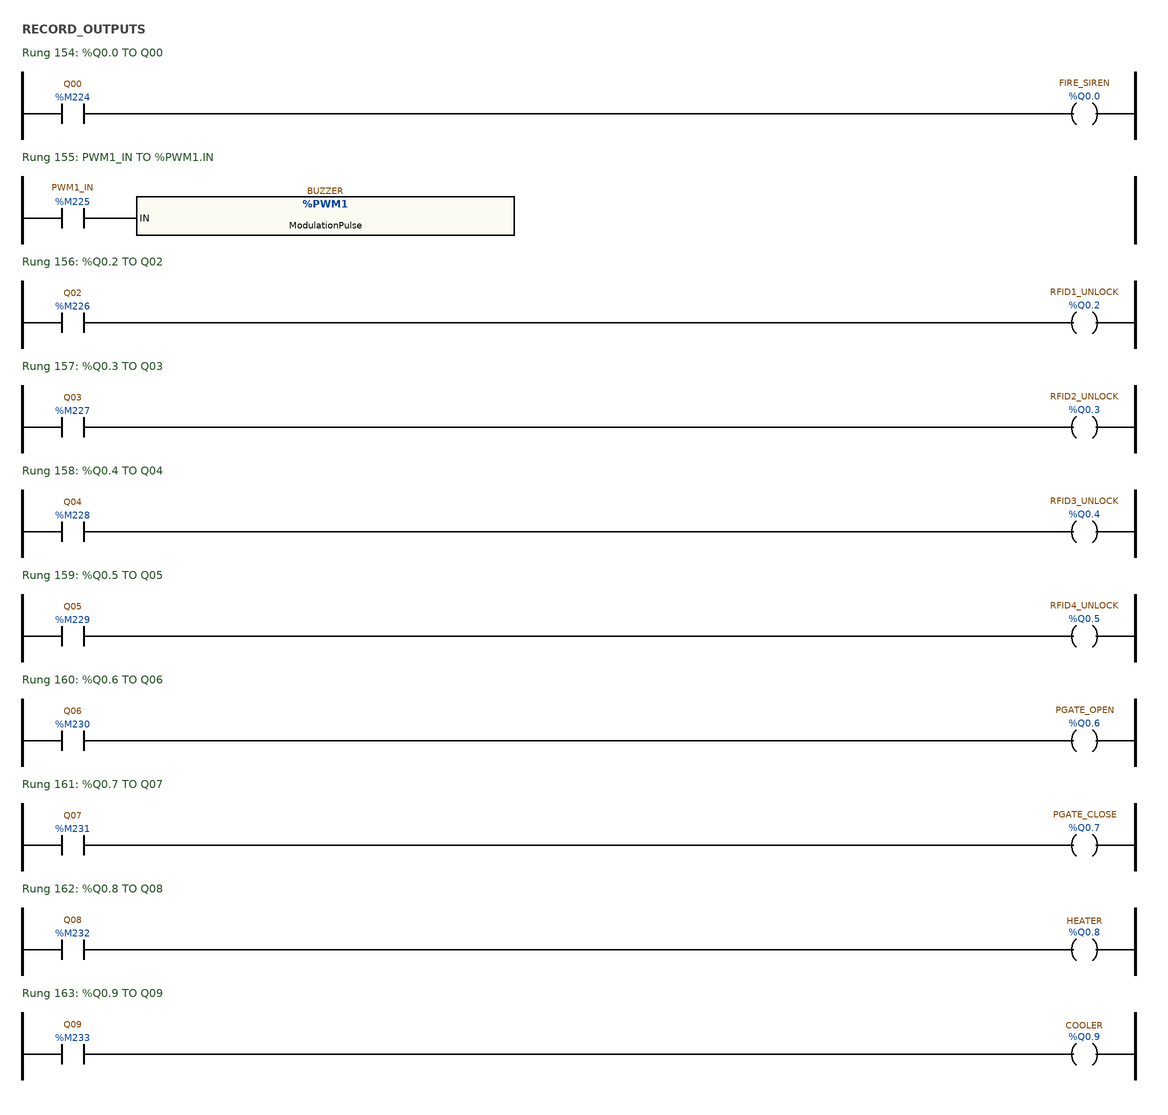

// Rung 154: %Q0.0 TO Q00
  LD %M224                (* Q00 *)
  ST %Q0.0                (* FIRE_SIREN *)
  // as ST:
  //   FIRE_SIREN := Q00;

// Rung 155: PWM1_IN TO %PWM1.IN
  BLK %PWM1               (* BUZZER *)
  LD %M225                (* PWM1_IN *)
  IN
  END_BLK
  // as ST:
  //   BUZZER(IN := PWM1_IN);

// Rung 156: %Q0.2 TO Q02
  LD %M226                (* Q02 *)
  ST %Q0.2                (* RFID1_UNLOCK *)
  // as ST:
  //   RFID1_UNLOCK := Q02;

// Rung 157: %Q0.3 TO Q03
  LD %M227                (* Q03 *)
  ST %Q0.3                (* RFID2_UNLOCK *)
  // as ST:
  //   RFID2_UNLOCK := Q03;

// Rung 158: %Q0.4 TO Q04
  LD %M228                (* Q04 *)
  ST %Q0.4                (* RFID3_UNLOCK *)
  // as ST:
  //   RFID3_UNLOCK := Q04;

// Rung 159: %Q0.5 TO Q05
  LD %M229                (* Q05 *)
  ST %Q0.5                (* RFID4_UNLOCK *)
  // as ST:
  //   RFID4_UNLOCK := Q05;

// Rung 160: %Q0.6 TO Q06
  LD %M230                (* Q06 *)
  ST %Q0.6                (* PGATE_OPEN *)
  // as ST:
  //   PGATE_OPEN := Q06;

// Rung 161: %Q0.7 TO Q07
  LD %M231                (* Q07 *)
  ST %Q0.7                (* PGATE_CLOSE *)
  // as ST:
  //   PGATE_CLOSE := Q07;

// Rung 162: %Q0.8 TO Q08
  LD %M232                (* Q08 *)
  ST %Q0.8                (* HEATER *)
  // as ST:
  //   HEATER := Q08;

// Rung 163: %Q0.9 TO Q09
  LD %M233                (* Q09 *)
  ST %Q0.9                (* COOLER *)
  // as ST:
  //   COOLER := Q09;

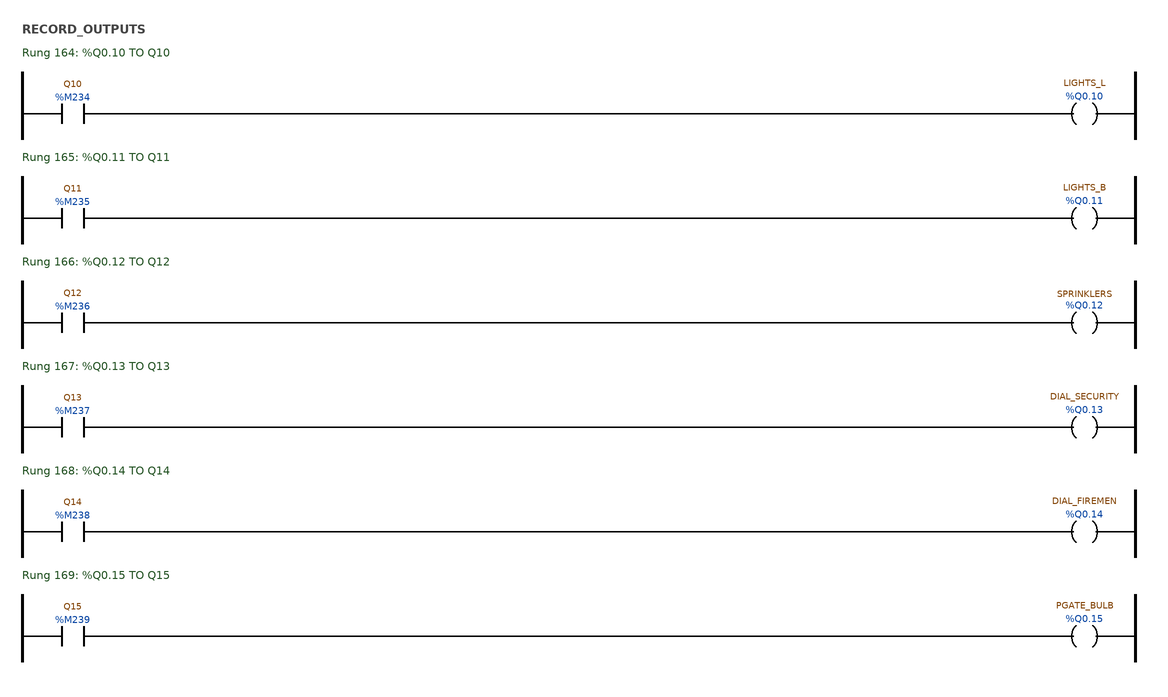

// Rung 164: %Q0.10 TO Q10
  LD %M234                (* Q10 *)
  ST %Q0.10               (* LIGHTS_L *)
  // as ST:
  //   LIGHTS_L := Q10;

// Rung 165: %Q0.11 TO Q11
  LD %M235                (* Q11 *)
  ST %Q0.11               (* LIGHTS_B *)
  // as ST:
  //   LIGHTS_B := Q11;

// Rung 166: %Q0.12 TO Q12
  LD %M236                (* Q12 *)
  ST %Q0.12               (* SPRINKLERS *)
  // as ST:
  //   SPRINKLERS := Q12;

// Rung 167: %Q0.13 TO Q13
  LD %M237                (* Q13 *)
  ST %Q0.13               (* DIAL_SECURITY *)
  // as ST:
  //   DIAL_SECURITY := Q13;

// Rung 168: %Q0.14 TO Q14
  LD %M238                (* Q14 *)
  ST %Q0.14               (* DIAL_FIREMEN *)
  // as ST:
  //   DIAL_FIREMEN := Q14;

// Rung 169: %Q0.15 TO Q15
  LD %M239                (* Q15 *)
  ST %Q0.15               (* PGATE_BULB *)
  // as ST:
  //   PGATE_BULB := Q15;
